LIN {X 0,Y 249.083,Z 81.458,A -85,B 0,C 180,E1 -19056.733,E2 -19056.733} C_VEL
LIN {X 0,Y 249.115,Z 81.452,A -85,B 0,C 180,E1 -19060.212,E2 -19060.212} C_VEL
LIN {X 0,Y 249.245,Z 81.417,A -85,B 0,C 180,E1 -19063.622,E2 -19063.622} C_VEL
LIN {X 0,Y 249.247,Z 81.438,A -85,B 0,C 180,E1 -19068.616,E2 -19068.616} C_VEL
LIN {X 0,Y 249.457,Z 81.409,A -85,B 0,C 180,E1 -19071.902,E2 -19071.902} C_VEL
LIN {X 0,Y 249.294,Z 81.412,A -85,B 0,C 180,E1 -19075.149,E2 -19075.149} C_VEL
LIN {X 0,Y 249.678,Z 81.38,A -85,B 0,C 180,E1 -19078.387,E2 -19078.387} C_VEL
LIN {X 0,Y 249.679,Z 81.385,A -85,B 0,C 180,E1 -19081.613,E2 -19081.613} C_VEL
LIN {X 0,Y 249.438,Z 81.412,A -85,B 0,C 180,E1 -19086.471,E2 -19086.471} C_VEL
LIN {X 0,Y 249.346,Z 81.422,A -85,B 0,C 180,E1 -19089.737,E2 -19089.737} C_VEL
LIN {X 0,Y 249.283,Z 81.427,A -85,B 0,C 180,E1 -19090.328,E2 -19090.328} C_VEL
LIN {X 0,Y 248.549,Z 81.525,A -85,B 0,C 180,E1 -19091.676,E2 -19091.676} C_VEL
LIN {X 0,Y 245.682,Z 81.88,A -85,B 0,C 180,E1 -19093.874,E2 -19093.874} C_VEL
LIN {X 0,Y 243.264,Z 82.181,A -85,B 0,C 180,E1 -19095.663,E2 -19095.663} C_VEL
LIN {X 0,Y 242.195,Z 82.315,A -85,B 0,C 180,E1 -19097.05,E2 -19097.05} C_VEL
LIN {X 0,Y 242.089,Z 82.325,A -85,B 0,C 180,E1 -19097.521,E2 -19097.521} C_VEL
LIN {X 0,Y 242.01,Z 82.339,A -85,B 0,C 180,E1 -19102.181,E2 -19102.181} C_VEL
LIN {X 0,Y 242.035,Z 82.335,A -85,B 0,C 180,E1 -19105.821,E2 -19105.821} C_VEL
LIN {X 0,Y 241.973,Z 82.344,A -85,B 0,C 180,E1 -19109.588,E2 -19109.588} C_VEL
LIN {X 0,Y 241.982,Z 82.343,A -85,B 0,C 180,E1 -19113.493,E2 -19113.493} C_VEL
LIN {X 0,Y 241.992,Z 82.341,A -85,B 0,C 180,E1 -19117.582,E2 -19117.582} C_VEL
LIN {X 0,Y 241.94,Z 82.348,A -85,B 0,C 180,E1 -19121.922,E2 -19121.922} C_VEL
LIN {X 0,Y 241.937,Z 82.351,A -85,B 0,C 180,E1 -19126.571,E2 -19126.571} C_VEL
LIN {X 0,Y 241.959,Z 82.347,A -85,B 0,C 180,E1 -19130.281,E2 -19130.281} C_VEL
LIN {X 0,Y 242.076,Z 82.527,A -85,B 0,C 180,E1 -19133.301,E2 -19133.301} C_VEL
LIN {X 0,Y 244.19,Z 91.874,A -85,B 0,C 180,E1 -19136.849,E2 -19136.849} C_VEL
LIN {X 0,Y 245.968,Z 100.654,A -85,B 0,C 180,E1 -19140.013,E2 -19140.013} C_VEL
LIN {X 0,Y 248.842,Z 109.122,A -85,B 0,C 180,E1 -19140.597,E2 -19140.597} C_VEL
LIN {X 0,Y 252.507,Z 138.269,A -85,B 0,C 180,E1 -19141.879,E2 -19141.879} C_VEL
LIN {X 0,Y 254.291,Z 157.169,A -85,B 0,C 180,E1 -19142.627,E2 -19142.627} C_VEL
LIN {X 0,Y 252.694,Z 210.32,A -85,B 0,C 180,E1 -19144.131,E2 -19144.131} C_VEL
LIN {X 0,Y 251.721,Z 223.453,A -85,B 0,C 180,E1 -19144.8,E2 -19144.8} C_VEL
LIN {X 0,Y 250.343,Z 236.124,A -85,B 0,C 180,E1 -19145.759,E2 -19145.759} C_VEL
LIN {X 0,Y 248.844,Z 247.387,A -85,B 0,C 180,E1 -19146.929,E2 -19146.929} C_VEL
LIN {X 0,Y 247.01,Z 259.074,A -85,B 0,C 180,E1 -19148.511,E2 -19148.511} C_VEL
LIN {X 0,Y 245.474,Z 268.522,A -85,B 0,C 180,E1 -19150.124,E2 -19150.124} C_VEL
LIN {X 0,Y 244.023,Z 276.962,A -85,B 0,C 180,E1 -19151.883,E2 -19151.883} C_VEL
LIN {X 0,Y 243.336,Z 280.982,A -85,B 0,C 180,E1 -19152.851,E2 -19152.851} C_VEL
LIN {X 0,Y 242.04,Z 289.578,A -85,B 0,C 180,E1 -19155.281,E2 -19155.281} C_VEL
LIN {X 0,Y 240.902,Z 296.619,A -85,B 0,C 180,E1 -19157.789,E2 -19157.789} C_VEL
LIN {X 0,Y 240.236,Z 303.085,A -85,B 0,C 180,E1 -19160.741,E2 -19160.741} C_VEL
LIN {X 0,Y 239.974,Z 307.313,A -85,B 0,C 180,E1 -19163.272,E2 -19163.272} C_VEL
LIN {X 0,Y 239.97,Z 309.546,A -85,B 0,C 180,E1 -19164.959,E2 -19164.959} C_VEL
LIN {X 0,Y 240.045,Z 311.282,A -85,B 0,C 180,E1 -19166.643,E2 -19166.643} C_VEL
LIN {X 0,Y 240.09,Z 312.593,A -85,B 0,C 180,E1 -19168.322,E2 -19168.322} C_VEL
LIN {X 0,Y 240.142,Z 313.499,A -85,B 0,C 180,E1 -19170,E2 -19170} C_VEL
LIN {X 0,Y 240.034,Z 313.985,A -85,B 0,C 180,E1 -19171.678,E2 -19171.678} C_VEL
LIN {X 0,Y 239.964,Z 314.036,A -85,B 0,C 180,E1 -19173.358,E2 -19173.358} C_VEL
LIN {X 0,Y 239.913,Z 313.67,A -85,B 0,C 180,E1 -19175.127,E2 -19175.127} C_VEL
LIN {X 0,Y 240.132,Z 311.863,A -85,B 0,C 180,E1 -19178.415,E2 -19178.415} C_VEL
LIN {X 0,Y 240.48,Z 310.31,A -85,B 0,C 180,E1 -19180.099,E2 -19180.099} C_VEL
LIN {X 0,Y 241.265,Z 307.21,A -85,B 0,C 180,E1 -19182.619,E2 -19182.619} C_VEL
LIN {X 0,Y 242.676,Z 303.085,A -85,B 0,C 180,E1 -19185.108,E2 -19185.108} C_VEL
LIN {X 0,Y 244.865,Z 296.801,A -85,B 0,C 180,E1 -19187.971,E2 -19187.971} C_VEL
LIN {X 0,Y 247.08,Z 289.994,A -85,B 0,C 180,E1 -19190.392,E2 -19190.392} C_VEL
LIN {X 0,Y 249.862,Z 281.575,A -85,B 0,C 180,E1 -19192.753,E2 -19192.753} C_VEL
LIN {X 0,Y 252.632,Z 272.932,A -85,B 0,C 180,E1 -19194.663,E2 -19194.663} C_VEL
LIN {X 0,Y 255.666,Z 262.319,A -85,B 0,C 180,E1 -19196.532,E2 -19196.532} C_VEL
LIN {X 0,Y 258.396,Z 251.803,A -85,B 0,C 180,E1 -19197.981,E2 -19197.981} C_VEL
LIN {X 0,Y 260.919,Z 240.172,A -85,B 0,C 180,E1 -19199.223,E2 -19199.223} C_VEL
LIN {X 0,Y 263.018,Z 228.115,A -85,B 0,C 180,E1 -19200.178,E2 -19200.178} C_VEL
LIN {X 0,Y 264.69,Z 214.429,A -85,B 0,C 180,E1 -19200.943,E2 -19200.943} C_VEL
LIN {X 0,Y 265.71,Z 200.941,A -85,B 0,C 180,E1 -19201.376,E2 -19201.376} C_VEL
LIN {X 0,Y 267.298,Z 160.216,A -85,B 0,C 180,E1 -19202.462,E2 -19202.462} C_VEL
LIN {X 0,Y 264.083,Z 138.448,A -85,B 0,C 180,E1 -19203.705,E2 -19203.705} C_VEL
LIN {X 0,Y 262.587,Z 131.019,A -85,B 0,C 180,E1 -19204.209,E2 -19204.209} C_VEL
LIN {X 0,Y 255.925,Z 116.639,A -85,B 0,C 180,E1 -19205.895,E2 -19205.895} C_VEL
LIN {X 0,Y 248.914,Z 103.116,A -85,B 0,C 180,E1 -19207.761,E2 -19207.761} C_VEL
LIN {X 0,Y 246.617,Z 98.7,A -85,B 0,C 180,E1 -19208.44,E2 -19208.44} C_VEL
LIN {X 0,Y 244.374,Z 90.616,A -85,B 0,C 180,E1 -19212.221,E2 -19212.221} C_VEL
LIN {X 0,Y 242.242,Z 83.517,A -85,B 0,C 180,E1 -19215.869,E2 -19215.869} C_VEL
LIN {X 0,Y 241.986,Z 82.334,A -85,B 0,C 180,E1 -19216.559,E2 -19216.559} C_VEL
LIN {X 0,Y 241.998,Z 82.337,A -85,B 0,C 180,E1 -19221.64,E2 -19221.64} C_VEL
LIN {X 0,Y 241.984,Z 82.339,A -85,B 0,C 180,E1 -19224.488,E2 -19224.488} C_VEL
LIN {X 0,Y 241.978,Z 82.344,A -85,B 0,C 180,E1 -19228.48,E2 -19228.48} C_VEL
LIN {X 0,Y 242.013,Z 82.34,A -85,B 0,C 180,E1 -19232.313,E2 -19232.313} C_VEL
LIN {X 0,Y 242.06,Z 82.333,A -85,B 0,C 180,E1 -19236.016,E2 -19236.016} C_VEL
LIN {X 0,Y 242.041,Z 82.33,A -85,B 0,C 180,E1 -19239.608,E2 -19239.608} C_VEL
LIN {X 0,Y 242.166,Z 82.307,A -85,B 0,C 180,E1 -19243.278,E2 -19243.278} C_VEL
LIN {X 0,Y 242.184,Z 82.304,A -85,B 0,C 180,E1 -19248.279,E2 -19248.279} C_VEL
LIN {X 0,Y 242.403,Z 82.284,A -85,B 0,C 180,E1 -19251.665,E2 -19251.665} C_VEL
LIN {X 0,Y 242.426,Z 82.271,A -85,B 0,C 180,E1 -19253.341,E2 -19253.341} C_VEL
LIN {X 0,Y 242.638,Z 82.246,A -85,B 0,C 180,E1 -19258.34,E2 -19258.34} C_VEL
LIN {X 0,Y 242.638,Z 82.26,A -85,B 0,C 180,E1 -19261.66,E2 -19261.66} C_VEL
LIN {X 0,Y 242.419,Z 82.288,A -85,B 0,C 180,E1 -19266.662,E2 -19266.662} C_VEL
LIN {X 0,Y 242.269,Z 82.298,A -85,B 0,C 180,E1 -19270.023,E2 -19270.023} C_VEL
LIN {X 0,Y 242.141,Z 82.315,A -85,B 0,C 180,E1 -19275.142,E2 -19275.142} C_VEL
LIN {X 0,Y 242.062,Z 82.321,A -85,B 0,C 180,E1 -19278.625,E2 -19278.625} C_VEL
LIN {X 0,Y 242.008,Z 82.333,A -85,B 0,C 180,E1 -19282.18,E2 -19282.18} C_VEL
LIN {X 0,Y 242.033,Z 82.335,A -85,B 0,C 180,E1 -19285.821,E2 -19285.821} C_VEL
LIN {X 0,Y 241.972,Z 82.343,A -85,B 0,C 180,E1 -19289.588,E2 -19289.588} C_VEL
LIN {X 0,Y 241.98,Z 82.338,A -85,B 0,C 180,E1 -19293.493,E2 -19293.493} C_VEL
LIN {X 0,Y 241.984,Z 82.339,A -85,B 0,C 180,E1 -19297.583,E2 -19297.583} C_VEL
LIN {X 0,Y 241.957,Z 82.325,A -85,B 0,C 180,E1 -19300.683,E2 -19300.683} C_VEL
LIN {X 0,Y 243.048,Z 85.314,A -85,B 0,C 180,E1 -19301.073,E2 -19301.073} C_VEL
LIN {X 0,Y 245.057,Z 87.692,A -85,B 0,C 180,E1 -19301.613,E2 -19301.613} C_VEL
LIN {X 0,Y 247.331,Z 91.154,A -85,B 0,C 180,E1 -19302.237,E2 -19302.237} C_VEL
LIN {X 0,Y 255.665,Z 104.188,A -85,B 0,C 180,E1 -19304.392,E2 -19304.392} C_VEL
LIN {X 0,Y 262.591,Z 116.027,A -85,B 0,C 180,E1 -19306.064,E2 -19306.064} C_VEL
LIN {X 0,Y 268.629,Z 128.906,A -85,B 0,C 180,E1 -19307.505,E2 -19307.505} C_VEL
LIN {X 0,Y 266.108,Z 185.116,A -85,B 0,C 180,E1 -19308.994,E2 -19308.994} C_VEL
LIN {X 0,Y 265.047,Z 197.91,A -85,B 0,C 180,E1 -19309.61,E2 -19309.61} C_VEL
LIN {X 0,Y 263.629,Z 209.846,A -85,B 0,C 180,E1 -19310.464,E2 -19310.464} C_VEL
LIN {X 0,Y 261.537,Z 222.38,A -85,B 0,C 180,E1 -19311.673,E2 -19311.673} C_VEL
LIN {X 0,Y 259.106,Z 233.731,A -85,B 0,C 180,E1 -19313.121,E2 -19313.121} C_VEL
LIN {X 0,Y 256.438,Z 244.411,A -85,B 0,C 180,E1 -19314.863,E2 -19314.863} C_VEL
LIN {X 0,Y 253.624,Z 253.941,A -85,B 0,C 180,E1 -19316.819,E2 -19316.819} C_VEL
LIN {X 0,Y 250.668,Z 263.079,A -85,B 0,C 180,E1 -19319.224,E2 -19319.224} C_VEL
LIN {X 0,Y 248.218,Z 269.982,A -85,B 0,C 180,E1 -19321.523,E2 -19321.523} C_VEL
LIN {X 0,Y 246.2,Z 275.278,A -85,B 0,C 180,E1 -19323.739,E2 -19323.739} C_VEL
LIN {X 0,Y 244.314,Z 279.989,A -85,B 0,C 180,E1 -19326.251,E2 -19326.251} C_VEL
LIN {X 0,Y 242.84,Z 283.543,A -85,B 0,C 180,E1 -19328.792,E2 -19328.792} C_VEL
LIN {X 0,Y 241.656,Z 286.048,A -85,B 0,C 180,E1 -19331.343,E2 -19331.343} C_VEL
LIN {X 0,Y 240.752,Z 287.793,A -85,B 0,C 180,E1 -19334.436,E2 -19334.436} C_VEL
LIN {X 0,Y 240.33,Z 288.182,A -85,B 0,C 180,E1 -19336.471,E2 -19336.471} C_VEL
LIN {X 0,Y 240.048,Z 288.099,A -85,B 0,C 180,E1 -19338.174,E2 -19338.174} C_VEL
LIN {X 0,Y 239.96,Z 287.599,A -85,B 0,C 180,E1 -19339.879,E2 -19339.879} C_VEL
LIN {X 0,Y 240.208,Z 285.348,A -85,B 0,C 180,E1 -19343.279,E2 -19343.279} C_VEL
LIN {X 0,Y 240.506,Z 282.58,A -85,B 0,C 180,E1 -19345.811,E2 -19345.811} C_VEL
LIN {X 0,Y 240.984,Z 278.805,A -85,B 0,C 180,E1 -19348.329,E2 -19348.329} C_VEL
LIN {X 0,Y 241.623,Z 273.927,A -85,B 0,C 180,E1 -19350.833,E2 -19350.833} C_VEL
LIN {X 0,Y 242.662,Z 267.78,A -85,B 0,C 180,E1 -19353.321,E2 -19353.321} C_VEL
LIN {X 0,Y 244.046,Z 260.126,A -85,B 0,C 180,E1 -19355.785,E2 -19355.785} C_VEL
LIN {X 0,Y 245.683,Z 250.533,A -85,B 0,C 180,E1 -19358.223,E2 -19358.223} C_VEL
LIN {X 0,Y 247.481,Z 240.605,A -85,B 0,C 180,E1 -19360.224,E2 -19360.224} C_VEL
LIN {X 0,Y 249.307,Z 229.377,A -85,B 0,C 180,E1 -19362,E2 -19362} C_VEL
LIN {X 0,Y 250.738,Z 218.415,A -85,B 0,C 180,E1 -19363.37,E2 -19363.37} C_VEL
LIN {X 0,Y 251.913,Z 206.317,A -85,B 0,C 180,E1 -19364.542,E2 -19364.542} C_VEL
LIN {X 0,Y 252.856,Z 193.622,A -85,B 0,C 180,E1 -19365.414,E2 -19365.414} C_VEL
LIN {X 0,Y 253.476,Z 180.26,A -85,B 0,C 180,E1 -19365.994,E2 -19365.994} C_VEL
LIN {X 0,Y 255.359,Z 113.557,A -85,B 0,C 180,E1 -19367.84,E2 -19367.84} C_VEL
LIN {X 0,Y 251.274,Z 102.48,A -85,B 0,C 180,E1 -19368.602,E2 -19368.602} C_VEL
LIN {X 0,Y 243.144,Z 85.322,A -85,B 0,C 180,E1 -19370.051,E2 -19370.051} C_VEL
LIN {X 0,Y 242.053,Z 82.327,A -85,B 0,C 180,E1 -19370.32,E2 -19370.32} C_VEL
LIN {X 0,Y 242.042,Z 82.334,A -85,B 0,C 180,E1 -19373.986,E2 -19373.986} C_VEL
LIN {X 0,Y 242.002,Z 82.341,A -85,B 0,C 180,E1 -19377.688,E2 -19377.688} C_VEL
LIN {X 0,Y 241.976,Z 82.341,A -85,B 0,C 180,E1 -19381.52,E2 -19381.52} C_VEL
LIN {X 0,Y 242.03,Z 82.338,A -85,B 0,C 180,E1 -19385.605,E2 -19385.605} C_VEL
LIN {X 0,Y 241.976,Z 82.344,A -85,B 0,C 180,E1 -19389.716,E2 -19389.716} C_VEL
LIN {X 0,Y 241.929,Z 82.346,A -85,B 0,C 180,E1 -19394.203,E2 -19394.203} C_VEL
LIN {X 0,Y 241.935,Z 82.345,A -85,B 0,C 180,E1 -19398.077,E2 -19398.077} C_VEL
LIN {X 0,Y 241.989,Z 82.339,A -85,B 0,C 180,E1 -19402.418,E2 -19402.418} C_VEL
LIN {X 0,Y 241.983,Z 82.34,A -85,B 0,C 180,E1 -19406.508,E2 -19406.508} C_VEL
LIN {X 0,Y 242.039,Z 82.332,A -85,B 0,C 180,E1 -19410.588,E2 -19410.588} C_VEL
LIN {X 0,Y 242.07,Z 82.329,A -85,B 0,C 180,E1 -19414.183,E2 -19414.183} C_VEL
LIN {X 0,Y 242.056,Z 82.334,A -85,B 0,C 180,E1 -19418.297,E2 -19418.297} C_VEL
LIN {X 0,Y 242.166,Z 82.298,A -85,B 0,C 180,E1 -19423.279,E2 -19423.279} C_VEL
LIN {X 0,Y 242.184,Z 82.317,A -85,B 0,C 180,E1 -19428.28,E2 -19428.28} C_VEL
LIN {X 0,Y 242.403,Z 82.288,A -85,B 0,C 180,E1 -19431.665,E2 -19431.665} C_VEL
LIN {X 0,Y 242.425,Z 82.278,A -85,B 0,C 180,E1 -19433.341,E2 -19433.341} C_VEL
LIN {X 0,Y 242.639,Z 82.255,A -85,B 0,C 180,E1 -19438.34,E2 -19438.34} C_VEL
LIN {X 0,Y 242.639,Z 82.262,A -85,B 0,C 180,E1 -19441.66,E2 -19441.66} C_VEL
LIN {X 0,Y 242.41,Z 82.288,A -85,B 0,C 180,E1 -19446.66,E2 -19446.66} C_VEL
LIN {X 0,Y 242.24,Z 82.305,A -85,B 0,C 180,E1 -19450.289,E2 -19450.289} C_VEL
LIN {X 0,Y 242.143,Z 82.321,A -85,B 0,C 180,E1 -19455.143,E2 -19455.143} C_VEL
LIN {X 0,Y 242.089,Z 82.325,A -85,B 0,C 180,E1 -19457.521,E2 -19457.521} C_VEL
LIN {X 0,Y 241.37,Z 82.42,A -85,B 0,C 180,E1 -19458.909,E2 -19458.909} C_VEL
LIN {X 0,Y 238.508,Z 82.777,A -85,B 0,C 180,E1 -19461.174,E2 -19461.174} C_VEL
LIN {X 0,Y 236.098,Z 83.079,A -85,B 0,C 180,E1 -19463.019,E2 -19463.019} C_VEL
LIN {X 0,Y 235.051,Z 83.206,A -85,B 0,C 180,E1 -19464.451,E2 -19464.451} C_VEL
LIN {X 0,Y 234.957,Z 83.216,A -85,B 0,C 180,E1 -19464.936,E2 -19464.936} C_VEL
LIN {X 0,Y 234.928,Z 83.222,A -85,B 0,C 180,E1 -19469.824,E2 -19469.824} C_VEL
LIN {X 0,Y 234.944,Z 83.221,A -85,B 0,C 180,E1 -19473.114,E2 -19473.114} C_VEL
LIN {X 0,Y 234.93,Z 83.223,A -85,B 0,C 180,E1 -19476.749,E2 -19476.749} C_VEL
LIN {X 0,Y 234.945,Z 83.219,A -85,B 0,C 180,E1 -19478.944,E2 -19478.944} C_VEL
LIN {X 0,Y 234.89,Z 83.224,A -85,B 0,C 180,E1 -19483.486,E2 -19483.486} C_VEL
LIN {X 0,Y 234.89,Z 83.229,A -85,B 0,C 180,E1 -19486.514,E2 -19486.514} C_VEL
LIN {X 0,Y 234.92,Z 83.224,A -85,B 0,C 180,E1 -19491.079,E2 -19491.079} C_VEL
LIN {X 0,Y 234.991,Z 83.34,A -85,B 0,C 180,E1 -19492.658,E2 -19492.658} C_VEL
LIN {X 0,Y 237.422,Z 93.969,A -85,B 0,C 180,E1 -19496.826,E2 -19496.826} C_VEL
LIN {X 0,Y 238.706,Z 100.362,A -85,B 0,C 180,E1 -19499.171,E2 -19499.171} C_VEL
LIN {X 0,Y 242.602,Z 111.238,A -85,B 0,C 180,E1 -19499.978,E2 -19499.978} C_VEL
LIN {X 0,Y 246.172,Z 140.741,A -85,B 0,C 180,E1 -19501.307,E2 -19501.307} C_VEL
LIN {X 0,Y 247.768,Z 157.118,A -85,B 0,C 180,E1 -19501.984,E2 -19501.984} C_VEL
LIN {X 0,Y 246.139,Z 209.645,A -85,B 0,C 180,E1 -19503.503,E2 -19503.503} C_VEL
LIN {X 0,Y 245.138,Z 222.877,A -85,B 0,C 180,E1 -19504.188,E2 -19504.188} C_VEL
LIN {X 0,Y 243.719,Z 235.602,A -85,B 0,C 180,E1 -19505.169,E2 -19505.169} C_VEL
LIN {X 0,Y 242.041,Z 247.703,A -85,B 0,C 180,E1 -19506.468,E2 -19506.468} C_VEL
LIN {X 0,Y 240.151,Z 259.261,A -85,B 0,C 180,E1 -19508.091,E2 -19508.091} C_VEL
LIN {X 0,Y 238.571,Z 268.612,A -85,B 0,C 180,E1 -19509.748,E2 -19509.748} C_VEL
LIN {X 0,Y 237,Z 277.213,A -85,B 0,C 180,E1 -19511.611,E2 -19511.611} C_VEL
LIN {X 0,Y 236.297,Z 281.517,A -85,B 0,C 180,E1 -19512.697,E2 -19512.697} C_VEL
LIN {X 0,Y 234.906,Z 290.102,A -85,B 0,C 180,E1 -19515.267,E2 -19515.267} C_VEL
LIN {X 0,Y 233.763,Z 296.97,A -85,B 0,C 180,E1 -19517.851,E2 -19517.851} C_VEL
LIN {X 0,Y 233.193,Z 302.47,A -85,B 0,C 180,E1 -19520.458,E2 -19520.458} C_VEL
LIN {X 0,Y 232.896,Z 306.752,A -85,B 0,C 180,E1 -19523.067,E2 -19523.067} C_VEL
LIN {X 0,Y 232.902,Z 309.02,A -85,B 0,C 180,E1 -19524.806,E2 -19524.806} C_VEL
LIN {X 0,Y 232.955,Z 310.795,A -85,B 0,C 180,E1 -19526.541,E2 -19526.541} C_VEL
LIN {X 0,Y 233.015,Z 312.131,A -85,B 0,C 180,E1 -19528.271,E2 -19528.271} C_VEL
LIN {X 0,Y 233.063,Z 313.059,A -85,B 0,C 180,E1 -19530,E2 -19530} C_VEL
LIN {X 0,Y 232.96,Z 313.578,A -85,B 0,C 180,E1 -19531.729,E2 -19531.729} C_VEL
LIN {X 0,Y 232.879,Z 313.662,A -85,B 0,C 180,E1 -19533.46,E2 -19533.46} C_VEL
LIN {X 0,Y 232.841,Z 313.344,A -85,B 0,C 180,E1 -19535.195,E2 -19535.195} C_VEL
LIN {X 0,Y 233.08,Z 311.558,A -85,B 0,C 180,E1 -19538.671,E2 -19538.671} C_VEL
LIN {X 0,Y 233.461,Z 310.048,A -85,B 0,C 180,E1 -19540.406,E2 -19540.406} C_VEL
LIN {X 0,Y 234.303,Z 306.995,A -85,B 0,C 180,E1 -19543.001,E2 -19543.001} C_VEL
LIN {X 0,Y 235.817,Z 302.92,A -85,B 0,C 180,E1 -19545.559,E2 -19545.559} C_VEL
LIN {X 0,Y 238.12,Z 296.696,A -85,B 0,C 180,E1 -19548.499,E2 -19548.499} C_VEL
LIN {X 0,Y 240.414,Z 289.955,A -85,B 0,C 180,E1 -19550.984,E2 -19550.984} C_VEL
LIN {X 0,Y 243.325,Z 281.632,A -85,B 0,C 180,E1 -19553.4,E2 -19553.4} C_VEL
LIN {X 0,Y 246.208,Z 273.103,A -85,B 0,C 180,E1 -19555.352,E2 -19555.352} C_VEL
LIN {X 0,Y 249.344,Z 262.609,A -85,B 0,C 180,E1 -19557.26,E2 -19557.26} C_VEL
LIN {X 0,Y 252.161,Z 252.24,A -85,B 0,C 180,E1 -19558.736,E2 -19558.736} C_VEL
LIN {X 0,Y 254.758,Z 240.886,A -85,B 0,C 180,E1 -19560.001,E2 -19560.001} C_VEL
LIN {X 0,Y 256.969,Z 229.22,A -85,B 0,C 180,E1 -19560.965,E2 -19560.965} C_VEL
LIN {X 0,Y 258.729,Z 215.521,A -85,B 0,C 180,E1 -19561.777,E2 -19561.777} C_VEL
LIN {X 0,Y 259.88,Z 202.343,A -85,B 0,C 180,E1 -19562.238,E2 -19562.238} C_VEL
LIN {X 0,Y 261.571,Z 161.244,A -85,B 0,C 180,E1 -19563.35,E2 -19563.35} C_VEL
LIN {X 0,Y 258.237,Z 138.412,A -85,B 0,C 180,E1 -19564.706,E2 -19564.706} C_VEL
LIN {X 0,Y 257.257,Z 134.015,A -85,B 0,C 180,E1 -19565.034,E2 -19565.034} C_VEL
LIN {X 0,Y 250.998,Z 120.403,A -85,B 0,C 180,E1 -19566.696,E2 -19566.696} C_VEL
LIN {X 0,Y 244.576,Z 107.852,A -85,B 0,C 180,E1 -19568.484,E2 -19568.484} C_VEL
LIN {X 0,Y 241.394,Z 102.28,A -85,B 0,C 180,E1 -19569.4,E2 -19569.4} C_VEL
LIN {X 0,Y 239.214,Z 98.113,A -85,B 0,C 180,E1 -19570.111,E2 -19570.111} C_VEL
LIN {X 0,Y 236.753,Z 89.25,A -85,B 0,C 180,E1 -19574.566,E2 -19574.566} C_VEL
LIN {X 0,Y 234.893,Z 83.215,A -85,B 0,C 180,E1 -19577.929,E2 -19577.929} C_VEL
LIN {X 0,Y 234.92,Z 83.213,A -85,B 0,C 180,E1 -19581.079,E2 -19581.079} C_VEL
LIN {X 0,Y 234.929,Z 83.216,A -85,B 0,C 180,E1 -19585.361,E2 -19585.361} C_VEL
LIN {X 0,Y 234.934,Z 83.213,A -85,B 0,C 180,E1 -19589.432,E2 -19589.432} C_VEL
LIN {X 0,Y 234.997,Z 83.202,A -85,B 0,C 180,E1 -19593.793,E2 -19593.793} C_VEL
LIN {X 0,Y 235.014,Z 83.2,A -85,B 0,C 180,E1 -19598.97,E2 -19598.97} C_VEL
LIN {X 0,Y 235.099,Z 83.186,A -85,B 0,C 180,E1 -19603.059,E2 -19603.059} C_VEL
LIN {X 0,Y 235.118,Z 83.183,A -85,B 0,C 180,E1 -19607.922,E2 -19607.922} C_VEL
LIN {X 0,Y 235.334,Z 83.167,A -85,B 0,C 180,E1 -19611.412,E2 -19611.412} C_VEL
LIN {X 0,Y 235.376,Z 83.149,A -85,B 0,C 180,E1 -19613.14,E2 -19613.14} C_VEL
LIN {X 0,Y 235.597,Z 83.122,A -85,B 0,C 180,E1 -19618.29,E2 -19618.29} C_VEL
LIN {X 0,Y 235.598,Z 83.136,A -85,B 0,C 180,E1 -19621.709,E2 -19621.709} C_VEL
LIN {X 0,Y 235.37,Z 83.167,A -85,B 0,C 180,E1 -19626.859,E2 -19626.859} C_VEL
LIN {X 0,Y 235.216,Z 83.179,A -85,B 0,C 180,E1 -19630.327,E2 -19630.327} C_VEL
LIN {X 0,Y 235.095,Z 83.197,A -85,B 0,C 180,E1 -19635.607,E2 -19635.607} C_VEL
LIN {X 0,Y 235.002,Z 83.201,A -85,B 0,C 180,E1 -19639.206,E2 -19639.206} C_VEL
LIN {X 0,Y 234.953,Z 83.208,A -85,B 0,C 180,E1 -19642.883,E2 -19642.883} C_VEL
LIN {X 0,Y 234.948,Z 83.21,A -85,B 0,C 180,E1 -19646.66,E2 -19646.66} C_VEL
LIN {X 0,Y 234.901,Z 83.217,A -85,B 0,C 180,E1 -19650.572,E2 -19650.572} C_VEL
LIN {X 0,Y 234.926,Z 83.217,A -85,B 0,C 180,E1 -19654.638,E2 -19654.638} C_VEL
LIN {X 0,Y 234.925,Z 83.216,A -85,B 0,C 180,E1 -19659.031,E2 -19659.031} C_VEL
LIN {X 0,Y 235.989,Z 86.175,A -85,B 0,C 180,E1 -19659.453,E2 -19659.453} C_VEL
LIN {X 0,Y 238.055,Z 88.413,A -85,B 0,C 180,E1 -19660.046,E2 -19660.046} C_VEL
LIN {X 0,Y 239.918,Z 91.502,A -85,B 0,C 180,E1 -19660.612,E2 -19660.612} C_VEL
LIN {X 0,Y 241.752,Z 94.11,A -85,B 0,C 180,E1 -19661.136,E2 -19661.136} C_VEL
LIN {X 0,Y 248.766,Z 104.769,A -85,B 0,C 180,E1 -19663.056,E2 -19663.056} C_VEL
LIN {X 0,Y 256.888,Z 118.447,A -85,B 0,C 180,E1 -19665.133,E2 -19665.133} C_VEL
LIN {X 0,Y 262.926,Z 131.138,A -85,B 0,C 180,E1 -19666.639,E2 -19666.639} C_VEL
LIN {X 0,Y 260.28,Z 186.314,A -85,B 0,C 180,E1 -19668.129,E2 -19668.129} C_VEL
LIN {X 0,Y 259.08,Z 199.617,A -85,B 0,C 180,E1 -19668.801,E2 -19668.801} C_VEL
LIN {X 0,Y 257.583,Z 211.623,A -85,B 0,C 180,E1 -19669.711,E2 -19669.711} C_VEL
LIN {X 0,Y 255.648,Z 222.43,A -85,B 0,C 180,E1 -19670.78,E2 -19670.78} C_VEL
LIN {X 0,Y 252.995,Z 234.347,A -85,B 0,C 180,E1 -19672.328,E2 -19672.328} C_VEL
LIN {X 0,Y 250.513,Z 243.897,A -85,B 0,C 180,E1 -19673.904,E2 -19673.904} C_VEL
LIN {X 0,Y 247.573,Z 253.623,A -85,B 0,C 180,E1 -19675.899,E2 -19675.899} C_VEL
LIN {X 0,Y 244.894,Z 261.521,A -85,B 0,C 180,E1 -19677.933,E2 -19677.933} C_VEL
LIN {X 0,Y 242.122,Z 269.178,A -85,B 0,C 180,E1 -19680.432,E2 -19680.432} C_VEL
LIN {X 0,Y 239.67,Z 275.284,A -85,B 0,C 180,E1 -19682.966,E2 -19682.966} C_VEL
LIN {X 0,Y 237.658,Z 280.076,A -85,B 0,C 180,E1 -19685.543,E2 -19685.543} C_VEL
LIN {X 0,Y 236.077,Z 283.706,A -85,B 0,C 180,E1 -19688.153,E2 -19688.153} C_VEL
LIN {X 0,Y 234.795,Z 286.284,A -85,B 0,C 180,E1 -19690.776,E2 -19690.776} C_VEL
LIN {X 0,Y 234.159,Z 287.477,A -85,B 0,C 180,E1 -19692.534,E2 -19692.534} C_VEL
LIN {X 0,Y 233.706,Z 288.219,A -85,B 0,C 180,E1 -19694.297,E2 -19694.297} C_VEL
LIN {X 0,Y 233.303,Z 288.555,A -85,B 0,C 180,E1 -19696.055,E2 -19696.055} C_VEL
LIN {X 0,Y 232.886,Z 288.062,A -85,B 0,C 180,E1 -19699.568,E2 -19699.568} C_VEL
LIN {X 0,Y 232.898,Z 287.179,A -85,B 0,C 180,E1 -19701.322,E2 -19701.322} C_VEL
LIN {X 0,Y 233.261,Z 285.191,A -85,B 0,C 180,E1 -19703.863,E2 -19703.863} C_VEL
LIN {X 0,Y 233.481,Z 282.097,A -85,B 0,C 180,E1 -19706.549,E2 -19706.549} C_VEL
LIN {X 0,Y 234.078,Z 278.038,A -85,B 0,C 180,E1 -19709.14,E2 -19709.14} C_VEL
LIN {X 0,Y 234.999,Z 271.83,A -85,B 0,C 180,E1 -19712.143,E2 -19712.143} C_VEL
LIN {X 0,Y 236.318,Z 265.058,A -85,B 0,C 180,E1 -19714.691,E2 -19714.691} C_VEL
LIN {X 0,Y 237.821,Z 256.654,A -85,B 0,C 180,E1 -19717.215,E2 -19717.215} C_VEL
LIN {X 0,Y 239.351,Z 248.004,A -85,B 0,C 180,E1 -19719.294,E2 -19719.294} C_VEL
LIN {X 0,Y 241.391,Z 237.309,A -85,B 0,C 180,E1 -19721.334,E2 -19721.334} C_VEL
LIN {X 0,Y 243.057,Z 226.683,A -85,B 0,C 180,E1 -19722.95,E2 -19722.95} C_VEL
LIN {X 0,Y 244.524,Z 214.816,A -85,B 0,C 180,E1 -19724.353,E2 -19724.353} C_VEL
LIN {X 0,Y 245.663,Z 202.504,A -85,B 0,C 180,E1 -19725.451,E2 -19725.451} C_VEL
LIN {X 0,Y 246.537,Z 189.774,A -85,B 0,C 180,E1 -19726.244,E2 -19726.244} C_VEL
LIN {X 0,Y 247.087,Z 175.916,A -85,B 0,C 180,E1 -19726.75,E2 -19726.75} C_VEL
LIN {X 0,Y 248.886,Z 115.206,A -85,B 0,C 180,E1 -19728.459,E2 -19728.459} C_VEL
LIN {X 0,Y 245.313,Z 105.535,A -85,B 0,C 180,E1 -19729.153,E2 -19729.153} C_VEL
LIN {X 0,Y 237.664,Z 89.241,A -85,B 0,C 180,E1 -19730.575,E2 -19730.575} C_VEL
LIN {X 0,Y 235.1,Z 83.875,A -85,B 0,C 180,E1 -19731.072,E2 -19731.072} C_VEL
LIN {X 0,Y 234.999,Z 83.205,A -85,B 0,C 180,E1 -19731.152,E2 -19731.152} C_VEL
LIN {X 0,Y 234.995,Z 83.214,A -85,B 0,C 180,E1 -19736.206,E2 -19736.206} C_VEL
LIN {X 0,Y 234.924,Z 83.22,A -85,B 0,C 180,E1 -19740.569,E2 -19740.569} C_VEL
LIN {X 0,Y 234.962,Z 83.216,A -85,B 0,C 180,E1 -19744.633,E2 -19744.633} C_VEL
LIN {X 0,Y 234.943,Z 83.218,A -85,B 0,C 180,E1 -19748.945,E2 -19748.945} C_VEL
LIN {X 0,Y 234.888,Z 83.227,A -85,B 0,C 180,E1 -19753.486,E2 -19753.486} C_VEL
LIN {X 0,Y 234.882,Z 83.223,A -85,B 0,C 180,E1 -19756.513,E2 -19756.513} C_VEL
LIN {X 0,Y 234.92,Z 83.219,A -85,B 0,C 180,E1 -19761.079,E2 -19761.079} C_VEL
LIN {X 0,Y 234.929,Z 83.219,A -85,B 0,C 180,E1 -19765.362,E2 -19765.362} C_VEL
LIN {X 0,Y 234.934,Z 83.215,A -85,B 0,C 180,E1 -19769.433,E2 -19769.433} C_VEL
LIN {X 0,Y 234.997,Z 83.21,A -85,B 0,C 180,E1 -19773.794,E2 -19773.794} C_VEL
LIN {X 0,Y 235.015,Z 83.209,A -85,B 0,C 180,E1 -19778.97,E2 -19778.97} C_VEL
LIN {X 0,Y 235.1,Z 83.177,A -85,B 0,C 180,E1 -19783.06,E2 -19783.06} C_VEL
LIN {X 0,Y 235.118,Z 83.195,A -85,B 0,C 180,E1 -19787.922,E2 -19787.922} C_VEL
LIN {X 0,Y 235.334,Z 83.168,A -85,B 0,C 180,E1 -19791.413,E2 -19791.413} C_VEL
LIN {X 0,Y 235.376,Z 83.156,A -85,B 0,C 180,E1 -19793.141,E2 -19793.141} C_VEL
LIN {X 0,Y 235.598,Z 83.131,A -85,B 0,C 180,E1 -19798.291,E2 -19798.291} C_VEL
LIN {X 0,Y 235.598,Z 83.14,A -85,B 0,C 180,E1 -19801.71,E2 -19801.71} C_VEL
LIN {X 0,Y 235.361,Z 83.166,A -85,B 0,C 180,E1 -19806.86,E2 -19806.86} C_VEL
LIN {X 0,Y 235.215,Z 83.18,A -85,B 0,C 180,E1 -19810.328,E2 -19810.328} C_VEL
LIN {X 0,Y 235.097,Z 83.198,A -85,B 0,C 180,E1 -19815.608,E2 -19815.608} C_VEL
LIN {X 0,Y 235.003,Z 83.211,A -85,B 0,C 180,E1 -19819.206,E2 -19819.206} C_VEL
LIN {X 0,Y 234.955,Z 83.22,A -85,B 0,C 180,E1 -19822.884,E2 -19822.884} C_VEL
LIN {X 0,Y 234.957,Z 83.216,A -85,B 0,C 180,E1 -19824.936,E2 -19824.936} C_VEL
LIN {X 0,Y 234.256,Z 83.306,A -85,B 0,C 180,E1 -19826.367,E2 -19826.367} C_VEL
LIN {X 0,Y 231.369,Z 83.667,A -85,B 0,C 180,E1 -19828.701,E2 -19828.701} C_VEL
LIN {X 0,Y 228.941,Z 83.97,A -85,B 0,C 180,E1 -19830.605,E2 -19830.605} C_VEL
LIN {X 0,Y 227.913,Z 84.097,A -85,B 0,C 180,E1 -19832.083,E2 -19832.083} C_VEL
LIN {X 0,Y 227.835,Z 84.101,A -85,B 0,C 180,E1 -19832.584,E2 -19832.584} C_VEL
LIN {X 0,Y 227.895,Z 84.1,A -85,B 0,C 180,E1 -19836.696,E2 -19836.696} C_VEL
LIN {X 0,Y 227.829,Z 84.108,A -85,B 0,C 180,E1 -19840.377,E2 -19840.377} C_VEL
LIN {X 0,Y 227.836,Z 84.104,A -85,B 0,C 180,E1 -19845.193,E2 -19845.193} C_VEL
LIN {X 0,Y 227.829,Z 84.108,A -85,B 0,C 180,E1 -19849.623,E2 -19849.623} C_VEL
LIN {X 0,Y 227.944,Z 84.265,A -85,B 0,C 180,E1 -19852.02,E2 -19852.02} C_VEL
LIN {X 0,Y 230.383,Z 94.817,A -85,B 0,C 180,E1 -19856.32,E2 -19856.32} C_VEL
LIN {X 0,Y 231.402,Z 99.861,A -85,B 0,C 180,E1 -19858.256,E2 -19858.256} C_VEL
LIN {X 0,Y 236.351,Z 113.094,A -85,B 0,C 180,E1 -19859.314,E2 -19859.314} C_VEL
LIN {X 0,Y 239.765,Z 142.084,A -85,B 0,C 180,E1 -19860.66,E2 -19860.66} C_VEL
LIN {X 0,Y 241.258,Z 158.328,A -85,B 0,C 180,E1 -19861.347,E2 -19861.347} C_VEL
LIN {X 0,Y 239.614,Z 208.938,A -85,B 0,C 180,E1 -19862.841,E2 -19862.841} C_VEL
LIN {X 0,Y 238.595,Z 222.285,A -85,B 0,C 180,E1 -19863.543,E2 -19863.543} C_VEL
LIN {X 0,Y 237.131,Z 235.067,A -85,B 0,C 180,E1 -19864.548,E2 -19864.548} C_VEL
LIN {X 0,Y 235.554,Z 246.424,A -85,B 0,C 180,E1 -19865.779,E2 -19865.779} C_VEL
LIN {X 0,Y 233.464,Z 258.128,A -85,B 0,C 180,E1 -19867.429,E2 -19867.429} C_VEL
LIN {X 0,Y 231.679,Z 268.702,A -85,B 0,C 180,E1 -19869.351,E2 -19869.351} C_VEL
LIN {X 0,Y 230.081,Z 277.151,A -85,B 0,C 180,E1 -19871.249,E2 -19871.249} C_VEL
LIN {X 0,Y 229.37,Z 280.655,A -85,B 0,C 180,E1 -19872.157,E2 -19872.157} C_VEL
LIN {X 0,Y 228.166,Z 288.037,A -85,B 0,C 180,E1 -19874.364,E2 -19874.364} C_VEL
LIN {X 0,Y 226.972,Z 295.274,A -85,B 0,C 180,E1 -19877.027,E2 -19877.027} C_VEL
LIN {X 0,Y 226.169,Z 301.857,A -85,B 0,C 180,E1 -19880.159,E2 -19880.159} C_VEL
LIN {X 0,Y 225.82,Z 306.19,A -85,B 0,C 180,E1 -19882.849,E2 -19882.849} C_VEL
LIN {X 0,Y 225.809,Z 308.73,A -85,B 0,C 180,E1 -19884.85,E2 -19884.85} C_VEL
LIN {X 0,Y 225.869,Z 310.309,A -85,B 0,C 180,E1 -19886.432,E2 -19886.432} C_VEL
LIN {X 0,Y 225.941,Z 311.668,A -85,B 0,C 180,E1 -19888.217,E2 -19888.217} C_VEL
LIN {X 0,Y 225.987,Z 312.619,A -85,B 0,C 180,E1 -19890,E2 -19890} C_VEL
LIN {X 0,Y 225.887,Z 313.162,A -85,B 0,C 180,E1 -19891.783,E2 -19891.783} C_VEL
LIN {X 0,Y 225.774,Z 313.084,A -85,B 0,C 180,E1 -19895.05,E2 -19895.05} C_VEL
LIN {X 0,Y 225.763,Z 312.31,A -85,B 0,C 180,E1 -19897.153,E2 -19897.153} C_VEL
LIN {X 0,Y 226.024,Z 311.249,A -85,B 0,C 180,E1 -19898.944,E2 -19898.944} C_VEL
LIN {X 0,Y 226.439,Z 309.784,A -85,B 0,C 180,E1 -19900.732,E2 -19900.732} C_VEL
LIN {X 0,Y 227.363,Z 306.772,A -85,B 0,C 180,E1 -19903.405,E2 -19903.405} C_VEL
LIN {X 0,Y 228.974,Z 302.746,A -85,B 0,C 180,E1 -19906.036,E2 -19906.036} C_VEL
LIN {X 0,Y 231.392,Z 296.601,A -85,B 0,C 180,E1 -19909.057,E2 -19909.057} C_VEL
LIN {X 0,Y 233.763,Z 289.925,A -85,B 0,C 180,E1 -19911.61,E2 -19911.61} C_VEL
LIN {X 0,Y 236.831,Z 281.675,A -85,B 0,C 180,E1 -19914.081,E2 -19914.081} C_VEL
LIN {X 0,Y 239.812,Z 273.259,A -85,B 0,C 180,E1 -19916.078,E2 -19916.078} C_VEL
LIN {X 0,Y 243.08,Z 262.899,A -85,B 0,C 180,E1 -19918.023,E2 -19918.023} C_VEL
LIN {X 0,Y 245.975,Z 252.676,A -85,B 0,C 180,E1 -19919.529,E2 -19919.529} C_VEL
LIN {X 0,Y 248.654,Z 241.52,A -85,B 0,C 180,E1 -19920.816,E2 -19920.816} C_VEL
LIN {X 0,Y 251.147,Z 229.038,A -85,B 0,C 180,E1 -19921.883,E2 -19921.883} C_VEL
LIN {X 0,Y 252.918,Z 215.886,A -85,B 0,C 180,E1 -19922.684,E2 -19922.684} C_VEL
LIN {X 0,Y 254.159,Z 202.363,A -85,B 0,C 180,E1 -19923.178,E2 -19923.178} C_VEL
LIN {X 0,Y 255.834,Z 161.301,A -85,B 0,C 180,E1 -19924.326,E2 -19924.326} C_VEL
LIN {X 0,Y 252.374,Z 137.934,A -85,B 0,C 180,E1 -19925.789,E2 -19925.789} C_VEL
LIN {X 0,Y 246.311,Z 124.511,A -85,B 0,C 180,E1 -19927.479,E2 -19927.479} C_VEL
LIN {X 0,Y 240.097,Z 112.246,A -85,B 0,C 180,E1 -19929.289,E2 -19929.289} C_VEL
LIN {X 0,Y 234.614,Z 102.494,A -85,B 0,C 180,E1 -19930.973,E2 -19930.973} C_VEL
LIN {X 0,Y 231.999,Z 98.038,A -85,B 0,C 180,E1 -19931.815,E2 -19931.815} C_VEL
LIN {X 0,Y 231.797,Z 97.488,A -85,B 0,C 180,E1 -19931.966,E2 -19931.966} C_VEL
LIN {X 0,Y 230.001,Z 91.127,A -85,B 0,C 180,E1 -19935.348,E2 -19935.348} C_VEL
LIN {X 0,Y 227.837,Z 84.093,A -85,B 0,C 180,E1 -19939.518,E2 -19939.518} C_VEL
LIN {X 0,Y 227.882,Z 84.091,A -85,B 0,C 180,E1 -19944.128,E2 -19944.128} C_VEL
LIN {X 0,Y 227.873,Z 84.1,A -85,B 0,C 180,E1 -19948.378,E2 -19948.378} C_VEL
LIN {X 0,Y 227.889,Z 84.098,A -85,B 0,C 180,E1 -19952.445,E2 -19952.445} C_VEL
LIN {X 0,Y 227.917,Z 84.096,A -85,B 0,C 180,E1 -19956.367,E2 -19956.367} C_VEL
LIN {X 0,Y 227.946,Z 84.09,A -85,B 0,C 180,E1 -19960.175,E2 -19960.175} C_VEL
LIN {X 0,Y 228.061,Z 84.066,A -85,B 0,C 180,E1 -19963.898,E2 -19963.898} C_VEL
LIN {X 0,Y 228.076,Z 84.061,A -85,B 0,C 180,E1 -19967.543,E2 -19967.543} C_VEL
LIN {X 0,Y 228.271,Z 84.05,A -85,B 0,C 180,E1 -19971.144,E2 -19971.144} C_VEL
LIN {X 0,Y 228.327,Z 84.027,A -85,B 0,C 180,E1 -19972.927,E2 -19972.927} C_VEL
LIN {X 0,Y 228.556,Z 83.999,A -85,B 0,C 180,E1 -19978.238,E2 -19978.238} C_VEL
LIN {X 0,Y 228.556,Z 84.012,A -85,B 0,C 180,E1 -19981.762,E2 -19981.762} C_VEL
LIN {X 0,Y 228.321,Z 84.042,A -85,B 0,C 180,E1 -19987.072,E2 -19987.072} C_VEL
LIN {X 0,Y 228.147,Z 84.064,A -85,B 0,C 180,E1 -19990.651,E2 -19990.651} C_VEL
LIN {X 0,Y 228.052,Z 84.064,A -85,B 0,C 180,E1 -19994.273,E2 -19994.273} C_VEL
LIN {X 0,Y 228,Z 84.074,A -85,B 0,C 180,E1 -19997.953,E2 -19997.953} C_VEL
LIN {X 0,Y 227.925,Z 84.085,A -85,B 0,C 180,E1 -20002.325,E2 -20002.325} C_VEL
LIN {X 0,Y 227.925,Z 84.085,A -85,B 0,C 180,E1 -20006.593,E2 -20006.593} C_VEL
LIN {X 0,Y 227.875,Z 84.093,A -85,B 0,C 180,E1 -20010.281,E2 -20010.281} C_VEL
LIN {X 0,Y 227.877,Z 84.093,A -85,B 0,C 180,E1 -20013.72,E2 -20013.72} C_VEL
LIN {X 0,Y 227.876,Z 84.198,A -85,B 0,C 180,E1 -20017.262,E2 -20017.262} C_VEL
LIN {X 0,Y 228.761,Z 86.793,A -85,B 0,C 180,E1 -20017.622,E2 -20017.622} C_VEL
LIN {X 0,Y 230.744,Z 88.982,A -85,B 0,C 180,E1 -20018.247,E2 -20018.247} C_VEL
LIN {X 0,Y 233.547,Z 93.094,A -85,B 0,C 180,E1 -20019.145,E2 -20019.145} C_VEL
LIN {X 0,Y 239.991,Z 102.481,A -85,B 0,C 180,E1 -20021.077,E2 -20021.077} C_VEL
LIN {X 0,Y 248.414,Z 115.987,A -85,B 0,C 180,E1 -20023.41,E2 -20023.41} C_VEL
LIN {X 0,Y 253.828,Z 125.97,A -85,B 0,C 180,E1 -20024.835,E2 -20024.835} C_VEL
LIN {X 0,Y 257.179,Z 133.207,A -85,B 0,C 180,E1 -20025.71,E2 -20025.71} C_VEL
LIN {X 0,Y 254.619,Z 186.261,A -85,B 0,C 180,E1 -20027.175,E2 -20027.175} C_VEL
LIN {X 0,Y 253.469,Z 199.007,A -85,B 0,C 180,E1 -20027.817,E2 -20027.817} C_VEL
LIN {X 0,Y 251.882,Z 211.186,A -85,B 0,C 180,E1 -20028.728,E2 -20028.728} C_VEL
LIN {X 0,Y 249.698,Z 223.11,A -85,B 0,C 180,E1 -20029.921,E2 -20029.921} C_VEL
LIN {X 0,Y 246.933,Z 234.964,A -85,B 0,C 180,E1 -20031.494,E2 -20031.494} C_VEL
LIN {X 0,Y 244.068,Z 245.45,A -85,B 0,C 180,E1 -20033.282,E2 -20033.282} C_VEL
LIN {X 0,Y 240.981,Z 255.004,A -85,B 0,C 180,E1 -20035.34,E2 -20035.34} C_VEL
LIN {X 0,Y 237.736,Z 264.09,A -85,B 0,C 180,E1 -20037.851,E2 -20037.851} C_VEL
LIN {X 0,Y 235.332,Z 270.27,A -85,B 0,C 180,E1 -20040.004,E2 -20040.004} C_VEL
LIN {X 0,Y 232.432,Z 277.074,A -85,B 0,C 180,E1 -20043.028,E2 -20043.028} C_VEL
LIN {X 0,Y 230.364,Z 281.662,A -85,B 0,C 180,E1 -20045.774,E2 -20045.774} C_VEL
LIN {X 0,Y 228.83,Z 284.88,A -85,B 0,C 180,E1 -20048.374,E2 -20048.374} C_VEL
LIN {X 0,Y 227.953,Z 286.522,A -85,B 0,C 180,E1 -20050.176,E2 -20050.176} C_VEL
LIN {X 0,Y 227.231,Z 287.751,A -85,B 0,C 180,E1 -20051.984,E2 -20051.984} C_VEL
LIN {X 0,Y 226.675,Z 288.604,A -85,B 0,C 180,E1 -20053.976,E2 -20053.976} C_VEL
LIN {X 0,Y 225.976,Z 288.911,A -85,B 0,C 180,E1 -20057.426,E2 -20057.426} C_VEL
LIN {X 0,Y 225.809,Z 288.505,A -85,B 0,C 180,E1 -20059.237,E2 -20059.237} C_VEL
LIN {X 0,Y 225.813,Z 287.684,A -85,B 0,C 180,E1 -20061.048,E2 -20061.048} C_VEL
LIN {X 0,Y 226.172,Z 285.522,A -85,B 0,C 180,E1 -20063.91,E2 -20063.91} C_VEL
LIN {X 0,Y 226.396,Z 282.727,A -85,B 0,C 180,E1 -20066.441,E2 -20066.441} C_VEL
LIN {X 0,Y 226.979,Z 278.744,A -85,B 0,C 180,E1 -20069.113,E2 -20069.113} C_VEL
LIN {X 0,Y 227.904,Z 272.634,A -85,B 0,C 180,E1 -20072.209,E2 -20072.209} C_VEL
LIN {X 0,Y 229.262,Z 265.952,A -85,B 0,C 180,E1 -20074.836,E2 -20074.836} C_VEL
LIN {X 0,Y 230.802,Z 257.692,A -85,B 0,C 180,E1 -20077.436,E2 -20077.436} C_VEL
LIN {X 0,Y 232.394,Z 249.19,A -85,B 0,C 180,E1 -20079.575,E2 -20079.575} C_VEL
LIN {X 0,Y 234.301,Z 239.822,A -85,B 0,C 180,E1 -20081.462,E2 -20081.462} C_VEL
LIN {X 0,Y 236.212,Z 228.243,A -85,B 0,C 180,E1 -20083.332,E2 -20083.332} C_VEL
LIN {X 0,Y 237.744,Z 216.811,A -85,B 0,C 180,E1 -20084.772,E2 -20084.772} C_VEL
LIN {X 0,Y 238.905,Z 205.009,A -85,B 0,C 180,E1 -20085.9,E2 -20085.9} C_VEL
LIN {X 0,Y 239.924,Z 191.365,A -85,B 0,C 180,E1 -20086.814,E2 -20086.814} C_VEL
LIN {X 0,Y 240.508,Z 177.857,A -85,B 0,C 180,E1 -20087.355,E2 -20087.355} C_VEL
LIN {X 0,Y 242.418,Z 116.804,A -85,B 0,C 180,E1 -20089.115,E2 -20089.115} C_VEL
LIN {X 0,Y 239.268,Z 108.327,A -85,B 0,C 180,E1 -20089.752,E2 -20089.752} C_VEL
LIN {X 0,Y 232,Z 92.831,A -85,B 0,C 180,E1 -20091.16,E2 -20091.16} C_VEL
LIN {X 0,Y 228.168,Z 85.142,A -85,B 0,C 180,E1 -20091.928,E2 -20091.928} C_VEL
LIN {X 0,Y 227.958,Z 84.087,A -85,B 0,C 180,E1 -20092.006,E2 -20092.006} C_VEL
LIN {X 0,Y 227.943,Z 84.092,A -85,B 0,C 180,E1 -20096.602,E2 -20096.602} C_VEL
LIN {X 0,Y 227.898,Z 84.096,A -85,B 0,C 180,E1 -20100.291,E2 -20100.291} C_VEL
LIN {X 0,Y 227.891,Z 84.097,A -85,B 0,C 180,E1 -20103.719,E2 -20103.719} C_VEL
LIN {X 0,Y 227.871,Z 84.1,A -85,B 0,C 180,E1 -20108.086,E2 -20108.086} C_VEL
LIN {X 0,Y 227.816,Z 84.105,A -85,B 0,C 180,E1 -20112.742,E2 -20112.742} C_VEL
LIN {X 0,Y 227.808,Z 84.107,A -85,B 0,C 180,E1 -20117.257,E2 -20117.257} C_VEL
LIN {X 0,Y 227.846,Z 84.101,A -85,B 0,C 180,E1 -20121.909,E2 -20121.909} C_VEL
LIN {X 0,Y 227.881,Z 84.096,A -85,B 0,C 180,E1 -20126.378,E2 -20126.378} C_VEL
LIN {X 0,Y 227.922,Z 84.089,A -85,B 0,C 180,E1 -20130.438,E2 -20130.438} C_VEL
LIN {X 0,Y 227.932,Z 84.09,A -85,B 0,C 180,E1 -20134.426,E2 -20134.426} C_VEL
LIN {X 0,Y 227.965,Z 84.089,A -85,B 0,C 180,E1 -20138.288,E2 -20138.288} C_VEL
LIN {X 0,Y 228.038,Z 84.057,A -85,B 0,C 180,E1 -20142.826,E2 -20142.826} C_VEL
LIN {X 0,Y 228.076,Z 84.07,A -85,B 0,C 180,E1 -20147.544,E2 -20147.544} C_VEL
LIN {X 0,Y 228.27,Z 84.047,A -85,B 0,C 180,E1 -20151.145,E2 -20151.145} C_VEL
LIN {X 0,Y 228.326,Z 84.033,A -85,B 0,C 180,E1 -20152.928,E2 -20152.928} C_VEL
LIN {X 0,Y 228.557,Z 84.006,A -85,B 0,C 180,E1 -20158.238,E2 -20158.238} C_VEL
LIN {X 0,Y 228.557,Z 84.017,A -85,B 0,C 180,E1 -20161.762,E2 -20161.762} C_VEL
LIN {X 0,Y 228.313,Z 84.045,A -85,B 0,C 180,E1 -20167.073,E2 -20167.073} C_VEL
LIN {X 0,Y 228.146,Z 84.06,A -85,B 0,C 180,E1 -20170.651,E2 -20170.651} C_VEL
LIN {X 0,Y 228.047,Z 84.075,A -85,B 0,C 180,E1 -20176.103,E2 -20176.103} C_VEL
LIN {X 0,Y 227.936,Z 84.088,A -85,B 0,C 180,E1 -20179.826,E2 -20179.826} C_VEL
LIN {X 0,Y 227.903,Z 84.096,A -85,B 0,C 180,E1 -20183.634,E2 -20183.634} C_VEL
LIN {X 0,Y 227.861,Z 84.102,A -85,B 0,C 180,E1 -20187.559,E2 -20187.559} C_VEL
LIN {X 0,Y 227.859,Z 84.103,A -85,B 0,C 180,E1 -20191.624,E2 -20191.624} C_VEL
LIN {X 0,Y 227.835,Z 84.101,A -85,B 0,C 180,E1 -20192.584,E2 -20192.584} C_VEL
LIN {X 0,Y 227.194,Z 84.186,A -85,B 0,C 180,E1 -20194.059,E2 -20194.059} C_VEL
LIN {X 0,Y 224.385,Z 84.539,A -85,B 0,C 180,E1 -20196.468,E2 -20196.468} C_VEL
LIN {X 0,Y 221.133,Z 84.943,A -85,B 0,C 180,E1 -20199.443,E2 -20199.443} C_VEL
LIN {X 0,Y 220.78,Z 84.983,A -85,B 0,C 180,E1 -20200.474,E2 -20200.474} C_VEL
LIN {X 0,Y 220.776,Z 84.986,A -85,B 0,C 180,E1 -20204.454,E2 -20204.454} C_VEL
LIN {X 0,Y 220.772,Z 84.986,A -85,B 0,C 180,E1 -20208.047,E2 -20208.047} C_VEL
LIN {X 0,Y 220.865,Z 85.136,A -85,B 0,C 180,E1 -20211.308,E2 -20211.308} C_VEL
LIN {X 0,Y 223.222,Z 94.912,A -85,B 0,C 180,E1 -20215.478,E2 -20215.478} C_VEL
LIN {X 0,Y 224.142,Z 99.598,A -85,B 0,C 180,E1 -20217.289,E2 -20217.289} C_VEL
LIN {X 0,Y 230.187,Z 115.591,A -85,B 0,C 180,E1 -20218.643,E2 -20218.643} C_VEL
LIN {X 0,Y 233.404,Z 143.471,A -85,B 0,C 180,E1 -20219.982,E2 -20219.982} C_VEL
LIN {X 0,Y 234.805,Z 158.198,A -85,B 0,C 180,E1 -20220.635,E2 -20220.635} C_VEL
LIN {X 0,Y 233.065,Z 209.341,A -85,B 0,C 180,E1 -20222.195,E2 -20222.195} C_VEL
LIN {X 0,Y 231.923,Z 223.191,A -85,B 0,C 180,E1 -20222.964,E2 -20222.964} C_VEL
LIN {X 0,Y 230.421,Z 235.598,A -85,B 0,C 180,E1 -20223.995,E2 -20223.995} C_VEL
LIN {X 0,Y 228.485,Z 248.301,A -85,B 0,C 180,E1 -20225.465,E2 -20225.465} C_VEL
LIN {X 0,Y 226.464,Z 259.609,A -85,B 0,C 180,E1 -20227.174,E2 -20227.174} C_VEL
LIN {X 0,Y 224.8,Z 268.773,A -85,B 0,C 180,E1 -20228.928,E2 -20228.928} C_VEL
LIN {X 0,Y 222.937,Z 277.982,A -85,B 0,C 180,E1 -20231.1,E2 -20231.1} C_VEL
LIN {X 0,Y 221.533,Z 285.881,A -85,B 0,C 180,E1 -20233.41,E2 -20233.41} C_VEL
LIN {X 0,Y 220.201,Z 293.445,A -85,B 0,C 180,E1 -20236.15,E2 -20236.15} C_VEL
LIN {X 0,Y 219.293,Z 299.511,A -85,B 0,C 180,E1 -20238.913,E2 -20238.913} C_VEL
LIN {X 0,Y 218.833,Z 304.3,A -85,B 0,C 180,E1 -20241.69,E2 -20241.69} C_VEL
LIN {X 0,Y 218.723,Z 308.474,A -85,B 0,C 180,E1 -20244.936,E2 -20244.936} C_VEL
LIN {X 0,Y 218.868,Z 311.205,A -85,B 0,C 180,E1 -20248.16,E2 -20248.16} C_VEL
LIN {X 0,Y 218.912,Z 312.178,A -85,B 0,C 180,E1 -20250,E2 -20250} C_VEL
LIN {X 0,Y 218.815,Z 312.744,A -85,B 0,C 180,E1 -20251.84,E2 -20251.84} C_VEL
LIN {X 0,Y 218.701,Z 312.764,A -85,B 0,C 180,E1 -20254.999,E2 -20254.999} C_VEL
LIN {X 0,Y 218.686,Z 311.98,A -85,B 0,C 180,E1 -20257.386,E2 -20257.386} C_VEL
LIN {X 0,Y 219.412,Z 309.514,A -85,B 0,C 180,E1 -20261.08,E2 -20261.08} C_VEL
LIN {X 0,Y 220.445,Z 306.541,A -85,B 0,C 180,E1 -20263.834,E2 -20263.834} C_VEL
LIN {X 0,Y 222.147,Z 302.566,A -85,B 0,C 180,E1 -20266.543,E2 -20266.543} C_VEL
LIN {X 0,Y 224.266,Z 297.479,A -85,B 0,C 180,E1 -20269.211,E2 -20269.211} C_VEL
LIN {X 0,Y 226.693,Z 291.123,A -85,B 0,C 180,E1 -20271.841,E2 -20271.841} C_VEL
LIN {X 0,Y 229.784,Z 283.206,A -85,B 0,C 180,E1 -20274.387,E2 -20274.387} C_VEL
LIN {X 0,Y 233.457,Z 273.389,A -85,B 0,C 180,E1 -20276.844,E2 -20276.844} C_VEL
LIN {X 0,Y 236.866,Z 263.189,A -85,B 0,C 180,E1 -20278.826,E2 -20278.826} C_VEL
LIN {X 0,Y 239.845,Z 253.112,A -85,B 0,C 180,E1 -20280.362,E2 -20280.362} C_VEL
LIN {X 0,Y 242.604,Z 242.153,A -85,B 0,C 180,E1 -20281.673,E2 -20281.673} C_VEL
LIN {X 0,Y 245.184,Z 230.026,A -85,B 0,C 180,E1 -20282.754,E2 -20282.754} C_VEL
LIN {X 0,Y 247.115,Z 216.923,A -85,B 0,C 180,E1 -20283.597,E2 -20283.597} C_VEL
LIN {X 0,Y 248.463,Z 203.403,A -85,B 0,C 180,E1 -20284.124,E2 -20284.124} C_VEL
LIN {X 0,Y 250.248,Z 162.448,A -85,B 0,C 180,E1 -20285.294,E2 -20285.294} C_VEL
LIN {X 0,Y 247.136,Z 140.859,A -85,B 0,C 180,E1 -20286.692,E2 -20286.692} C_VEL
LIN {X 0,Y 240.614,Z 126.274,A -85,B 0,C 180,E1 -20288.612,E2 -20288.612} C_VEL
LIN {X 0,Y 235.31,Z 115.989,A -85,B 0,C 180,E1 -20290.237,E2 -20290.237} C_VEL
LIN {X 0,Y 230.412,Z 107.192,A -85,B 0,C 180,E1 -20291.818,E2 -20291.818} C_VEL
LIN {X 0,Y 227.25,Z 101.961,A -85,B 0,C 180,E1 -20292.881,E2 -20292.881} C_VEL
LIN {X 0,Y 224.644,Z 97.525,A -85,B 0,C 180,E1 -20293.802,E2 -20293.802} C_VEL
LIN {X 0,Y 224.411,Z 97.01,A -85,B 0,C 180,E1 -20293.92,E2 -20293.92} C_VEL
LIN {X 0,Y 222.497,Z 90.484,A -85,B 0,C 180,E1 -20297.697,E2 -20297.697} C_VEL
LIN {X 0,Y 220.787,Z 84.975,A -85,B 0,C 180,E1 -20301.268,E2 -20301.268} C_VEL
LIN {X 0,Y 220.809,Z 84.971,A -85,B 0,C 180,E1 -20305.847,E2 -20305.847} C_VEL
LIN {X 0,Y 220.87,Z 84.965,A -85,B 0,C 180,E1 -20309.395,E2 -20309.395} C_VEL
LIN {X 0,Y 220.898,Z 84.959,A -85,B 0,C 180,E1 -20313.55,E2 -20313.55} C_VEL
LIN {X 0,Y 220.881,Z 84.961,A -85,B 0,C 180,E1 -20317.553,E2 -20317.553} C_VEL
LIN {X 0,Y 220.987,Z 84.944,A -85,B 0,C 180,E1 -20322.571,E2 -20322.571} C_VEL
LIN {X 0,Y 221.015,Z 84.942,A -85,B 0,C 180,E1 -20327.138,E2 -20327.138} C_VEL
LIN {X 0,Y 221.208,Z 84.93,A -85,B 0,C 180,E1 -20330.859,E2 -20330.859} C_VEL
LIN {X 0,Y 221.262,Z 84.907,A -85,B 0,C 180,E1 -20332.7,E2 -20332.7} C_VEL
LIN {X 0,Y 221.514,Z 84.876,A -85,B 0,C 180,E1 -20338.182,E2 -20338.182} C_VEL
LIN {X 0,Y 221.514,Z 84.889,A -85,B 0,C 180,E1 -20341.818,E2 -20341.818} C_VEL
LIN {X 0,Y 221.256,Z 84.919,A -85,B 0,C 180,E1 -20347.299,E2 -20347.299} C_VEL
LIN {X 0,Y 221.068,Z 84.947,A -85,B 0,C 180,E1 -20350.996,E2 -20350.996} C_VEL
LIN {X 0,Y 221.008,Z 84.957,A -85,B 0,C 180,E1 -20356.63,E2 -20356.63} C_VEL
LIN {X 0,Y 220.886,Z 84.97,A -85,B 0,C 180,E1 -20360.487,E2 -20360.487} C_VEL
LIN {X 0,Y 220.853,Z 84.971,A -85,B 0,C 180,E1 -20364.437,E2 -20364.437} C_VEL
LIN {X 0,Y 220.807,Z 84.979,A -85,B 0,C 180,E1 -20368.518,E2 -20368.518} C_VEL
LIN {X 0,Y 220.813,Z 84.979,A -85,B 0,C 180,E1 -20372.757,E2 -20372.757} C_VEL
LIN {X 0,Y 220.827,Z 84.977,A -85,B 0,C 180,E1 -20375.229,E2 -20375.229} C_VEL
LIN {X 0,Y 221.774,Z 87.742,A -85,B 0,C 180,E1 -20375.682,E2 -20375.682} C_VEL
LIN {X 0,Y 223.935,Z 89.977,A -85,B 0,C 180,E1 -20376.424,E2 -20376.424} C_VEL
LIN {X 0,Y 226.442,Z 93.883,A -85,B 0,C 180,E1 -20377.314,E2 -20377.314} C_VEL
LIN {X 0,Y 227.779,Z 95.52,A -85,B 0,C 180,E1 -20377.753,E2 -20377.753} C_VEL
LIN {X 0,Y 234.065,Z 104.655,A -85,B 0,C 180,E1 -20379.769,E2 -20379.769} C_VEL
LIN {X 0,Y 240.842,Z 115.361,A -85,B 0,C 180,E1 -20381.788,E2 -20381.788} C_VEL
LIN {X 0,Y 248.081,Z 127.978,A -85,B 0,C 180,E1 -20383.796,E2 -20383.796} C_VEL
LIN {X 0,Y 251.596,Z 135.566,A -85,B 0,C 180,E1 -20384.763,E2 -20384.763} C_VEL
LIN {X 0,Y 248.938,Z 187.371,A -85,B 0,C 180,E1 -20386.223,E2 -20386.223} C_VEL
LIN {X 0,Y 247.647,Z 200.568,A -85,B 0,C 180,E1 -20386.917,E2 -20386.917} C_VEL
LIN {X 0,Y 245.96,Z 212.811,A -85,B 0,C 180,E1 -20387.881,E2 -20387.881} C_VEL
LIN {X 0,Y 243.809,Z 223.79,A -85,B 0,C 180,E1 -20389.02,E2 -20389.02} C_VEL
LIN {X 0,Y 240.926,Z 235.583,A -85,B 0,C 180,E1 -20390.62,E2 -20390.62} C_VEL
LIN {X 0,Y 237.816,Z 246.457,A -85,B 0,C 180,E1 -20392.525,E2 -20392.525} C_VEL
LIN {X 0,Y 234.433,Z 256.362,A -85,B 0,C 180,E1 -20394.754,E2 -20394.754} C_VEL
LIN {X 0,Y 231.069,Z 265.283,A -85,B 0,C 180,E1 -20397.325,E2 -20397.325} C_VEL
LIN {X 0,Y 228.491,Z 271.521,A -85,B 0,C 180,E1 -20399.612,E2 -20399.612} C_VEL
LIN {X 0,Y 225.958,Z 277.121,A -85,B 0,C 180,E1 -20402.19,E2 -20402.19} C_VEL
LIN {X 0,Y 223.811,Z 281.667,A -85,B 0,C 180,E1 -20404.918,E2 -20404.918} C_VEL
LIN {X 0,Y 222.088,Z 285.084,A -85,B 0,C 180,E1 -20407.682,E2 -20407.682} C_VEL
LIN {X 0,Y 221.117,Z 286.762,A -85,B 0,C 180,E1 -20409.536,E2 -20409.536} C_VEL
LIN {X 0,Y 220.33,Z 288.025,A -85,B 0,C 180,E1 -20411.399,E2 -20411.399} C_VEL
LIN {X 0,Y 219.646,Z 289.009,A -85,B 0,C 180,E1 -20413.721,E2 -20413.721} C_VEL
LIN {X 0,Y 218.96,Z 289.316,A -85,B 0,C 180,E1 -20417.016,E2 -20417.016} C_VEL
LIN {X 0,Y 218.713,Z 288.18,A -85,B 0,C 180,E1 -20420.754,E2 -20420.754} C_VEL
LIN {X 0,Y 219.081,Z 285.844,A -85,B 0,C 180,E1 -20423.968,E2 -20423.968} C_VEL
LIN {X 0,Y 219.413,Z 282.138,A -85,B 0,C 180,E1 -20427.246,E2 -20427.246} C_VEL
LIN {X 0,Y 220.117,Z 277.863,A -85,B 0,C 180,E1 -20430,E2 -20430} C_VEL
LIN {X 0,Y 221.259,Z 271.412,A -85,B 0,C 180,E1 -20433.187,E2 -20433.187} C_VEL
LIN {X 0,Y 222.719,Z 264.325,A -85,B 0,C 180,E1 -20435.887,E2 -20435.887} C_VEL
LIN {X 0,Y 224.432,Z 255.519,A -85,B 0,C 180,E1 -20438.554,E2 -20438.554} C_VEL
LIN {X 0,Y 226.173,Z 246.489,A -85,B 0,C 180,E1 -20440.745,E2 -20440.745} C_VEL
LIN {X 0,Y 228.201,Z 236.457,A -85,B 0,C 180,E1 -20442.676,E2 -20442.676} C_VEL
LIN {X 0,Y 230.012,Z 225.342,A -85,B 0,C 180,E1 -20444.375,E2 -20444.375} C_VEL
LIN {X 0,Y 231.581,Z 212.929,A -85,B 0,C 180,E1 -20445.851,E2 -20445.851} C_VEL
LIN {X 0,Y 232.81,Z 200.233,A -85,B 0,C 180,E1 -20446.948,E2 -20446.948} C_VEL
LIN {X 0,Y 233.681,Z 186.643,A -85,B 0,C 180,E1 -20447.734,E2 -20447.734} C_VEL
LIN {X 0,Y 235.497,Z 135.916,A -85,B 0,C 180,E1 -20449.278,E2 -20449.278} C_VEL
LIN {X 0,Y 235.89,Z 117.953,A -85,B 0,C 180,E1 -20449.831,E2 -20449.831} C_VEL
LIN {X 0,Y 231.555,Z 107.213,A -85,B 0,C 180,E1 -20450.723,E2 -20450.723} C_VEL
LIN {X 0,Y 223.49,Z 90.807,A -85,B 0,C 180,E1 -20452.367,E2 -20452.367} C_VEL
LIN {X 0,Y 221.075,Z 86.003,A -85,B 0,C 180,E1 -20452.884,E2 -20452.884} C_VEL
LIN {X 0,Y 220.875,Z 84.97,A -85,B 0,C 180,E1 -20452.984,E2 -20452.984} C_VEL
LIN {X 0,Y 220.884,Z 84.971,A -85,B 0,C 180,E1 -20457.015,E2 -20457.015} C_VEL
LIN {X 0,Y 220.839,Z 84.973,A -85,B 0,C 180,E1 -20460.768,E2 -20460.768} C_VEL
LIN {X 0,Y 220.817,Z 84.978,A -85,B 0,C 180,E1 -20464.953,E2 -20464.953} C_VEL
LIN {X 0,Y 220.84,Z 84.974,A -85,B 0,C 180,E1 -20467.288,E2 -20467.288} C_VEL
LIN {X 0,Y 220.778,Z 84.982,A -85,B 0,C 180,E1 -20471.951,E2 -20471.951} C_VEL
LIN {X 0,Y 220.772,Z 84.98,A -85,B 0,C 180,E1 -20475.546,E2 -20475.546} C_VEL
LIN {X 0,Y 220.808,Z 84.974,A -85,B 0,C 180,E1 -20480.464,E2 -20480.464} C_VEL
LIN {X 0,Y 220.803,Z 84.976,A -85,B 0,C 180,E1 -20485.046,E2 -20485.046} C_VEL
LIN {X 0,Y 220.87,Z 84.967,A -85,B 0,C 180,E1 -20489.395,E2 -20489.395} C_VEL
LIN {X 0,Y 220.898,Z 84.966,A -85,B 0,C 180,E1 -20493.55,E2 -20493.55} C_VEL
LIN {X 0,Y 220.881,Z 84.97,A -85,B 0,C 180,E1 -20497.554,E2 -20497.554} C_VEL
LIN {X 0,Y 220.988,Z 84.935,A -85,B 0,C 180,E1 -20502.571,E2 -20502.571} C_VEL
LIN {X 0,Y 221.015,Z 84.95,A -85,B 0,C 180,E1 -20507.139,E2 -20507.139} C_VEL
LIN {X 0,Y 221.208,Z 84.927,A -85,B 0,C 180,E1 -20510.86,E2 -20510.86} C_VEL
LIN {X 0,Y 221.262,Z 84.913,A -85,B 0,C 180,E1 -20512.701,E2 -20512.701} C_VEL
LIN {X 0,Y 221.514,Z 84.882,A -85,B 0,C 180,E1 -20518.182,E2 -20518.182} C_VEL
LIN {X 0,Y 221.514,Z 84.893,A -85,B 0,C 180,E1 -20521.818,E2 -20521.818} C_VEL
LIN {X 0,Y 221.25,Z 84.925,A -85,B 0,C 180,E1 -20527.3,E2 -20527.3} C_VEL
LIN {X 0,Y 221.066,Z 84.943,A -85,B 0,C 180,E1 -20530.997,E2 -20530.997} C_VEL
LIN {X 0,Y 221.01,Z 84.952,A -85,B 0,C 180,E1 -20536.631,E2 -20536.631} C_VEL
LIN {X 0,Y 220.888,Z 84.966,A -85,B 0,C 180,E1 -20540.487,E2 -20540.487} C_VEL
LIN {X 0,Y 220.854,Z 84.974,A -85,B 0,C 180,E1 -20544.437,E2 -20544.437} C_VEL
LIN {X 0,Y 220.809,Z 84.982,A -85,B 0,C 180,E1 -20548.518,E2 -20548.518} C_VEL
LIN {X 0,Y 220.815,Z 84.982,A -85,B 0,C 180,E1 -20552.757,E2 -20552.757} C_VEL
LIN {X 0,Y 220.813,Z 84.98,A -85,B 0,C 180,E1 -20557.278,E2 -20557.278} C_VEL
LIN {X 0,Y 220.78,Z 84.983,A -85,B 0,C 180,E1 -20560.474,E2 -20560.474} C_VEL
LIN {X 0,Y 220.044,Z 85.077,A -85,B 0,C 180,E1 -20561.994,E2 -20561.994} C_VEL
LIN {X 0,Y 217.124,Z 85.441,A -85,B 0,C 180,E1 -20564.475,E2 -20564.475} C_VEL
LIN {X 0,Y 214.715,Z 85.741,A -85,B 0,C 180,E1 -20566.501,E2 -20566.501} C_VEL
LIN {X 0,Y 213.743,Z 85.861,A -85,B 0,C 180,E1 -20568.076,E2 -20568.076} C_VEL
LIN {X 0,Y 213.694,Z 85.867,A -85,B 0,C 180,E1 -20568.609,E2 -20568.609} C_VEL
LIN {X 0,Y 213.78,Z 85.867,A -85,B 0,C 180,E1 -20570.486,E2 -20570.486} C_VEL
LIN {X 0,Y 215.927,Z 94.779,A -85,B 0,C 180,E1 -20574.46,E2 -20574.46} C_VEL
LIN {X 0,Y 216.883,Z 99.186,A -85,B 0,C 180,E1 -20576.243,E2 -20576.243} C_VEL
LIN {X 0,Y 223.989,Z 117.453,A -85,B 0,C 180,E1 -20577.905,E2 -20577.905} C_VEL
LIN {X 0,Y 227.006,Z 144.157,A -85,B 0,C 180,E1 -20579.232,E2 -20579.232} C_VEL
LIN {X 0,Y 228.345,Z 159.528,A -85,B 0,C 180,E1 -20579.927,E2 -20579.927} C_VEL
LIN {X 0,Y 226.606,Z 208.265,A -85,B 0,C 180,E1 -20581.44,E2 -20581.44} C_VEL
LIN {X 0,Y 225.509,Z 221.795,A -85,B 0,C 180,E1 -20582.192,E2 -20582.192} C_VEL
LIN {X 0,Y 224.063,Z 233.948,A -85,B 0,C 180,E1 -20583.199,E2 -20583.199} C_VEL
LIN {X 0,Y 222.35,Z 245.403,A -85,B 0,C 180,E1 -20584.49,E2 -20584.49} C_VEL
LIN {X 0,Y 220.099,Z 257.156,A -85,B 0,C 180,E1 -20586.226,E2 -20586.226} C_VEL
LIN {X 0,Y 218.132,Z 267.761,A -85,B 0,C 180,E1 -20588.252,E2 -20588.252} C_VEL
LIN {X 0,Y 216.23,Z 277.115,A -85,B 0,C 180,E1 -20590.489,E2 -20590.489} C_VEL
LIN {X 0,Y 215.385,Z 281.023,A -85,B 0,C 180,E1 -20591.585,E2 -20591.585} C_VEL
LIN {X 0,Y 213.956,Z 289.125,A -85,B 0,C 180,E1 -20594.276,E2 -20594.276} C_VEL
LIN {X 0,Y 212.675,Z 295.964,A -85,B 0,C 180,E1 -20597.111,E2 -20597.111} C_VEL
LIN {X 0,Y 211.907,Z 302.249,A -85,B 0,C 180,E1 -20600.454,E2 -20600.454} C_VEL
LIN {X 0,Y 211.641,Z 306.317,A -85,B 0,C 180,E1 -20603.326,E2 -20603.326} C_VEL
LIN {X 0,Y 211.667,Z 309.309,A -85,B 0,C 180,E1 -20606.192,E2 -20606.192} C_VEL
LIN {X 0,Y 211.795,Z 310.74,A -85,B 0,C 180,E1 -20608.098,E2 -20608.098} C_VEL
LIN {X 0,Y 211.84,Z 311.737,A -85,B 0,C 180,E1 -20610,E2 -20610} C_VEL
LIN {X 0,Y 211.743,Z 312.325,A -85,B 0,C 180,E1 -20611.902,E2 -20611.902} C_VEL
LIN {X 0,Y 211.606,Z 312.422,A -85,B 0,C 180,E1 -20614.873,E2 -20614.873} C_VEL
LIN {X 0,Y 211.625,Z 311.651,A -85,B 0,C 180,E1 -20617.634,E2 -20617.634} C_VEL
LIN {X 0,Y 212.402,Z 309.233,A -85,B 0,C 180,E1 -20621.451,E2 -20621.451} C_VEL
LIN {X 0,Y 213.515,Z 306.308,A -85,B 0,C 180,E1 -20624.292,E2 -20624.292} C_VEL
LIN {X 0,Y 215.317,Z 302.384,A -85,B 0,C 180,E1 -20627.083,E2 -20627.083} C_VEL
LIN {X 0,Y 217.557,Z 297.354,A -85,B 0,C 180,E1 -20629.828,E2 -20629.828} C_VEL
LIN {X 0,Y 220.082,Z 291.067,A -85,B 0,C 180,E1 -20632.532,E2 -20632.532} C_VEL
LIN {X 0,Y 223.338,Z 283.251,A -85,B 0,C 180,E1 -20635.139,E2 -20635.139} C_VEL
LIN {X 0,Y 227.16,Z 273.523,A -85,B 0,C 180,E1 -20637.651,E2 -20637.651} C_VEL
LIN {X 0,Y 230.69,Z 263.485,A -85,B 0,C 180,E1 -20639.674,E2 -20639.674} C_VEL
LIN {X 0,Y 233.771,Z 253.565,A -85,B 0,C 180,E1 -20641.238,E2 -20641.238} C_VEL
LIN {X 0,Y 236.612,Z 242.812,A -85,B 0,C 180,E1 -20642.572,E2 -20642.572} C_VEL
LIN {X 0,Y 239.499,Z 229.853,A -85,B 0,C 180,E1 -20643.76,E2 -20643.76} C_VEL
LIN {X 0,Y 241.462,Z 217.203,A -85,B 0,C 180,E1 -20644.597,E2 -20644.597} C_VEL
LIN {X 0,Y 242.845,Z 204.531,A -85,B 0,C 180,E1 -20645.113,E2 -20645.113} C_VEL
LIN {X 0,Y 244.741,Z 163.589,A -85,B 0,C 180,E1 -20646.308,E2 -20646.308} C_VEL
LIN {X 0,Y 241.998,Z 144.011,A -85,B 0,C 180,E1 -20647.617,E2 -20647.617} C_VEL
LIN {X 0,Y 236.014,Z 130.356,A -85,B 0,C 180,E1 -20649.475,E2 -20649.475} C_VEL
LIN {X 0,Y 230.821,Z 120.081,A -85,B 0,C 180,E1 -20651.152,E2 -20651.152} C_VEL
LIN {X 0,Y 226.215,Z 111.773,A -85,B 0,C 180,E1 -20652.713,E2 -20652.713} C_VEL
LIN {X 0,Y 223.061,Z 106.483,A -85,B 0,C 180,E1 -20653.828,E2 -20653.828} C_VEL
LIN {X 0,Y 219.905,Z 101.278,A -85,B 0,C 180,E1 -20655,E2 -20655} C_VEL
LIN {X 0,Y 217.255,Z 96.977,A -85,B 0,C 180,E1 -20656.03,E2 -20656.03} C_VEL
LIN {X 0,Y 216.996,Z 96.336,A -85,B 0,C 180,E1 -20656.202,E2 -20656.202} C_VEL
LIN {X 0,Y 214.956,Z 89.742,A -85,B 0,C 180,E1 -20660.39,E2 -20660.39} C_VEL
LIN {X 0,Y 213.756,Z 85.846,A -85,B 0,C 180,E1 -20663.144,E2 -20663.144} C_VEL
LIN {X 0,Y 213.759,Z 85.848,A -85,B 0,C 180,E1 -20666.018,E2 -20666.018} C_VEL
LIN {X 0,Y 213.783,Z 85.845,A -85,B 0,C 180,E1 -20670.454,E2 -20670.454} C_VEL
LIN {X 0,Y 213.804,Z 85.843,A -85,B 0,C 180,E1 -20674.702,E2 -20674.702} C_VEL
LIN {X 0,Y 213.815,Z 85.839,A -85,B 0,C 180,E1 -20678.803,E2 -20678.803} C_VEL
LIN {X 0,Y 213.947,Z 85.82,A -85,B 0,C 180,E1 -20682.804,E2 -20682.804} C_VEL
LIN {X 0,Y 213.956,Z 85.824,A -85,B 0,C 180,E1 -20686.707,E2 -20686.707} C_VEL
LIN {X 0,Y 214.145,Z 85.811,A -85,B 0,C 180,E1 -20690.555,E2 -20690.555} C_VEL
LIN {X 0,Y 214.102,Z 85.804,A -85,B 0,C 180,E1 -20694.348,E2 -20694.348} C_VEL
LIN {X 0,Y 214.447,Z 85.756,A -85,B 0,C 180,E1 -20698.122,E2 -20698.122} C_VEL
LIN {X 0,Y 214.553,Z 85.753,A -85,B 0,C 180,E1 -20700,E2 -20700} C_VEL
LIN {X 0,Y 214.447,Z 85.769,A -85,B 0,C 180,E1 -20701.878,E2 -20701.878} C_VEL
LIN {X 0,Y 214.196,Z 85.796,A -85,B 0,C 180,E1 -20707.541,E2 -20707.541} C_VEL
LIN {X 0,Y 213.999,Z 85.83,A -85,B 0,C 180,E1 -20711.364,E2 -20711.364} C_VEL
LIN {X 0,Y 213.922,Z 85.83,A -85,B 0,C 180,E1 -20715.238,E2 -20715.238} C_VEL
LIN {X 0,Y 213.835,Z 85.837,A -85,B 0,C 180,E1 -20719.188,E2 -20719.188} C_VEL
LIN {X 0,Y 213.806,Z 85.841,A -85,B 0,C 180,E1 -20723.232,E2 -20723.232} C_VEL
LIN {X 0,Y 213.789,Z 85.845,A -85,B 0,C 180,E1 -20727.428,E2 -20727.428} C_VEL
LIN {X 0,Y 213.759,Z 85.854,A -85,B 0,C 180,E1 -20731.739,E2 -20731.739} C_VEL
LIN {X 0,Y 213.769,Z 85.854,A -85,B 0,C 180,E1 -20732.992,E2 -20732.992} C_VEL
LIN {X 0,Y 214.764,Z 88.713,A -85,B 0,C 180,E1 -20733.519,E2 -20733.519} C_VEL
LIN {X 0,Y 216.86,Z 90.878,A -85,B 0,C 180,E1 -20734.318,E2 -20734.318} C_VEL
LIN {X 0,Y 217.537,Z 91.697,A -85,B 0,C 180,E1 -20734.576,E2 -20734.576} C_VEL
LIN {X 0,Y 219.729,Z 94.976,A -85,B 0,C 180,E1 -20735.421,E2 -20735.421} C_VEL
LIN {X 0,Y 221.09,Z 96.643,A -85,B 0,C 180,E1 -20735.912,E2 -20735.912} C_VEL
LIN {X 0,Y 223.535,Z 100.032,A -85,B 0,C 180,E1 -20736.787,E2 -20736.787} C_VEL
LIN {X 0,Y 230.066,Z 109.596,A -85,B 0,C 180,E1 -20738.983,E2 -20738.983} C_VEL
LIN {X 0,Y 237.809,Z 122.032,A -85,B 0,C 180,E1 -20741.378,E2 -20741.378} C_VEL
LIN {X 0,Y 244.163,Z 133.63,A -85,B 0,C 180,E1 -20743.215,E2 -20743.215} C_VEL
LIN {X 0,Y 246.083,Z 137.813,A -85,B 0,C 180,E1 -20743.767,E2 -20743.767} C_VEL
LIN {X 0,Y 243.421,Z 187.511,A -85,B 0,C 180,E1 -20745.186,E2 -20745.186} C_VEL
LIN {X 0,Y 242.064,Z 200.888,A -85,B 0,C 180,E1 -20745.897,E2 -20745.897} C_VEL
LIN {X 0,Y 240.343,Z 212.841,A -85,B 0,C 180,E1 -20746.845,E2 -20746.845} C_VEL
LIN {X 0,Y 237.978,Z 224.485,A -85,B 0,C 180,E1 -20748.074,E2 -20748.074} C_VEL
LIN {X 0,Y 234.978,Z 236.221,A -85,B 0,C 180,E1 -20749.7,E2 -20749.7} C_VEL
LIN {X 0,Y 231.832,Z 246.728,A -85,B 0,C 180,E1 -20751.577,E2 -20751.577} C_VEL
LIN {X 0,Y 228.491,Z 256.184,A -85,B 0,C 180,E1 -20753.729,E2 -20753.729} C_VEL
LIN {X 0,Y 224.949,Z 265.108,A -85,B 0,C 180,E1 -20756.32,E2 -20756.32} C_VEL
LIN {X 0,Y 221.986,Z 272.025,A -85,B 0,C 180,E1 -20758.896,E2 -20758.896} C_VEL
LIN {X 0,Y 219.541,Z 277.141,A -85,B 0,C 180,E1 -20761.303,E2 -20761.303} C_VEL
LIN {X 0,Y 217.222,Z 281.781,A -85,B 0,C 180,E1 -20764.101,E2 -20764.101} C_VEL
LIN {X 0,Y 215.384,Z 285.272,A -85,B 0,C 180,E1 -20766.948,E2 -20766.948} C_VEL
LIN {X 0,Y 214.314,Z 287.002,A -85,B 0,C 180,E1 -20768.855,E2 -20768.855} C_VEL
LIN {X 0,Y 212.828,Z 289.192,A -85,B 0,C 180,E1 -20772.711,E2 -20772.711} C_VEL
LIN {X 0,Y 212.315,Z 289.675,A -85,B 0,C 180,E1 -20774.644,E2 -20774.644} C_VEL
LIN {X 0,Y 211.686,Z 289.383,A -85,B 0,C 180,E1 -20778.51,E2 -20778.51} C_VEL
LIN {X 0,Y 211.637,Z 288.654,A -85,B 0,C 180,E1 -20780.442,E2 -20780.442} C_VEL
LIN {X 0,Y 211.996,Z 286.181,A -85,B 0,C 180,E1 -20784.013,E2 -20784.013} C_VEL
LIN {X 0,Y 212.316,Z 282.777,A -85,B 0,C 180,E1 -20787.154,E2 -20787.154} C_VEL
LIN {X 0,Y 213.024,Z 278.577,A -85,B 0,C 180,E1 -20790,E2 -20790} C_VEL
LIN {X 0,Y 214.154,Z 272.215,A -85,B 0,C 180,E1 -20793.293,E2 -20793.293} C_VEL
LIN {X 0,Y 215.672,Z 265.261,A -85,B 0,C 180,E1 -20796.08,E2 -20796.08} C_VEL
LIN {X 0,Y 217.43,Z 256.57,A -85,B 0,C 180,E1 -20798.832,E2 -20798.832} C_VEL
LIN {X 0,Y 219.241,Z 247.669,A -85,B 0,C 180,E1 -20801.089,E2 -20801.089} C_VEL
LIN {X 0,Y 221.333,Z 237.839,A -85,B 0,C 180,E1 -20803.076,E2 -20803.076} C_VEL
LIN {X 0,Y 223.211,Z 227.013,A -85,B 0,C 180,E1 -20804.823,E2 -20804.823} C_VEL
LIN {X 0,Y 224.862,Z 214.921,A -85,B 0,C 180,E1 -20806.338,E2 -20806.338} C_VEL
LIN {X 0,Y 226.169,Z 202.282,A -85,B 0,C 180,E1 -20807.52,E2 -20807.52} C_VEL
LIN {X 0,Y 227.09,Z 189.389,A -85,B 0,C 180,E1 -20808.336,E2 -20808.336} C_VEL
LIN {X 0,Y 227.813,Z 171.418,A -85,B 0,C 180,E1 -20808.979,E2 -20808.979} C_VEL
LIN {X 0,Y 229.581,Z 119.779,A -85,B 0,C 180,E1 -20810.539,E2 -20810.539} C_VEL
LIN {X 0,Y 223.94,Z 106.505,A -85,B 0,C 180,E1 -20811.742,E2 -20811.742} C_VEL
LIN {X 0,Y 216.661,Z 92.07,A -85,B 0,C 180,E1 -20813.307,E2 -20813.307} C_VEL
LIN {X 0,Y 214.052,Z 86.954,A -85,B 0,C 180,E1 -20813.896,E2 -20813.896} C_VEL
LIN {X 0,Y 213.841,Z 85.846,A -85,B 0,C 180,E1 -20813.992,E2 -20813.992} C_VEL
LIN {X 0,Y 213.83,Z 85.85,A -85,B 0,C 180,E1 -20817.45,E2 -20817.45} C_VEL
LIN {X 0,Y 213.771,Z 85.855,A -85,B 0,C 180,E1 -20821.737,E2 -20821.737} C_VEL
LIN {X 0,Y 213.754,Z 85.858,A -85,B 0,C 180,E1 -20826.287,E2 -20826.287} C_VEL
LIN {X 0,Y 213.719,Z 85.859,A -85,B 0,C 180,E1 -20831.124,E2 -20831.124} C_VEL
LIN {X 0,Y 213.708,Z 85.863,A -85,B 0,C 180,E1 -20833.679,E2 -20833.679} C_VEL
LIN {X 0,Y 213.704,Z 85.861,A -85,B 0,C 180,E1 -20836.345,E2 -20836.345} C_VEL
LIN {X 0,Y 213.718,Z 85.859,A -85,B 0,C 180,E1 -20839.144,E2 -20839.144} C_VEL
LIN {X 0,Y 213.745,Z 85.854,A -85,B 0,C 180,E1 -20843.712,E2 -20843.712} C_VEL
LIN {X 0,Y 213.797,Z 85.85,A -85,B 0,C 180,E1 -20848.725,E2 -20848.725} C_VEL
LIN {X 0,Y 213.828,Z 85.85,A -85,B 0,C 180,E1 -20852.604,E2 -20852.604} C_VEL
LIN {X 0,Y 213.855,Z 85.847,A -85,B 0,C 180,E1 -20856.953,E2 -20856.953} C_VEL
LIN {X 0,Y 213.947,Z 85.81,A -85,B 0,C 180,E1 -20862.804,E2 -20862.804} C_VEL
LIN {X 0,Y 213.956,Z 85.826,A -85,B 0,C 180,E1 -20866.707,E2 -20866.707} C_VEL
LIN {X 0,Y 214.145,Z 85.808,A -85,B 0,C 180,E1 -20870.556,E2 -20870.556} C_VEL
LIN {X 0,Y 214.1,Z 85.792,A -85,B 0,C 180,E1 -20874.349,E2 -20874.349} C_VEL
LIN {X 0,Y 214.447,Z 85.761,A -85,B 0,C 180,E1 -20878.122,E2 -20878.122} C_VEL
LIN {X 0,Y 214.554,Z 85.758,A -85,B 0,C 180,E1 -20880,E2 -20880} C_VEL
LIN {X 0,Y 214.447,Z 85.773,A -85,B 0,C 180,E1 -20881.878,E2 -20881.878} C_VEL
LIN {X 0,Y 214.191,Z 85.806,A -85,B 0,C 180,E1 -20887.542,E2 -20887.542} C_VEL
LIN {X 0,Y 213.997,Z 85.825,A -85,B 0,C 180,E1 -20891.365,E2 -20891.365} C_VEL
LIN {X 0,Y 213.92,Z 85.835,A -85,B 0,C 180,E1 -20895.238,E2 -20895.238} C_VEL
LIN {X 0,Y 213.837,Z 85.848,A -85,B 0,C 180,E1 -20899.188,E2 -20899.188} C_VEL
LIN {X 0,Y 213.807,Z 85.854,A -85,B 0,C 180,E1 -20903.232,E2 -20903.232} C_VEL
LIN {X 0,Y 213.791,Z 85.856,A -85,B 0,C 180,E1 -20907.429,E2 -20907.429} C_VEL
LIN {X 0,Y 213.761,Z 85.859,A -85,B 0,C 180,E1 -20911.739,E2 -20911.739} C_VEL
LIN {X 0,Y 213.747,Z 85.862,A -85,B 0,C 180,E1 -20916.288,E2 -20916.288} C_VEL
LIN {X 0,Y 213.715,Z 85.864,A -85,B 0,C 180,E1 -20921.125,E2 -20921.125} C_VEL
LIN {X 0,Y 213.709,Z 85.863,A -85,B 0,C 180,E1 -20923.678,E2 -20923.678} C_VEL
LIN {X 0,Y 213.709,Z 85.866,A -85,B 0,C 180,E1 -20926.344,E2 -20926.344} C_VEL
LIN {X 0,Y 213.694,Z 85.867,A -85,B 0,C 180,E1 -20928.609,E2 -20928.609} C_VEL
LIN {X 0,Y 213.184,Z 86.46,A -85,B 0,C 180,E1 -20929.644,E2 -20929.644} C_VEL
LIN {X 0,Y 211.943,Z 87.907,A -85,B 0,C 180,E1 -20930.599,E2 -20930.599} C_VEL
LIN {X 0,Y 208.926,Z 92.946,A -85,B 0,C 180,E1 -20932.685,E2 -20932.685} C_VEL
LIN {X 0,Y 208.764,Z 95.217,A -85,B 0,C 180,E1 -20933.626,E2 -20933.626} C_VEL
LIN {X 0,Y 209.561,Z 98.57,A -85,B 0,C 180,E1 -20935.098,E2 -20935.098} C_VEL
LIN {X 0,Y 217.829,Z 119.516,A -85,B 0,C 180,E1 -20937.134,E2 -20937.134} C_VEL
LIN {X 0,Y 220.662,Z 144.988,A -85,B 0,C 180,E1 -20938.449,E2 -20938.449} C_VEL
LIN {X 0,Y 221.953,Z 159.719,A -85,B 0,C 180,E1 -20939.143,E2 -20939.143} C_VEL
LIN {X 0,Y 220.119,Z 208.687,A -85,B 0,C 180,E1 -20940.715,E2 -20940.715} C_VEL
LIN {X 0,Y 218.983,Z 221.936,A -85,B 0,C 180,E1 -20941.484,E2 -20941.484} C_VEL
LIN {X 0,Y 217.41,Z 234.507,A -85,B 0,C 180,E1 -20942.571,E2 -20942.571} C_VEL
LIN {X 0,Y 215.64,Z 245.697,A -85,B 0,C 180,E1 -20943.897,E2 -20943.897} C_VEL
LIN {X 0,Y 213.314,Z 257.32,A -85,B 0,C 180,E1 -20945.68,E2 -20945.68} C_VEL
LIN {X 0,Y 211.285,Z 267.833,A -85,B 0,C 180,E1 -20947.767,E2 -20947.767} C_VEL
LIN {X 0,Y 209.347,Z 277.003,A -85,B 0,C 180,E1 -20950.051,E2 -20950.051} C_VEL
LIN {X 0,Y 208.53,Z 279.88,A -85,B 0,C 180,E1 -20950.87,E2 -20950.87} C_VEL
LIN {X 0,Y 207.564,Z 285.691,A -85,B 0,C 180,E1 -20952.766,E2 -20952.766} C_VEL
LIN {X 0,Y 206.13,Z 293.153,A -85,B 0,C 180,E1 -20955.688,E2 -20955.688} C_VEL
LIN {X 0,Y 205.046,Z 299.992,A -85,B 0,C 180,E1 -20959.134,E2 -20959.134} C_VEL
LIN {X 0,Y 204.619,Z 304.494,A -85,B 0,C 180,E1 -20962.103,E2 -20962.103} C_VEL
LIN {X 0,Y 204.559,Z 307.925,A -85,B 0,C 180,E1 -20965.107,E2 -20965.107} C_VEL
LIN {X 0,Y 204.699,Z 310.274,A -85,B 0,C 180,E1 -20968.032,E2 -20968.032} C_VEL
LIN {X 0,Y 204.769,Z 311.296,A -85,B 0,C 180,E1 -20970,E2 -20970} C_VEL
LIN {X 0,Y 204.672,Z 311.907,A -85,B 0,C 180,E1 -20971.968,E2 -20971.968} C_VEL
LIN {X 0,Y 204.539,Z 312.072,A -85,B 0,C 180,E1 -20974.829,E2 -20974.829} C_VEL
LIN {X 0,Y 204.582,Z 311.323,A -85,B 0,C 180,E1 -20977.898,E2 -20977.898} C_VEL
LIN {X 0,Y 205.412,Z 308.95,A -85,B 0,C 180,E1 -20981.846,E2 -20981.846} C_VEL
LIN {X 0,Y 206.612,Z 306.075,A -85,B 0,C 180,E1 -20984.78,E2 -20984.78} C_VEL
LIN {X 0,Y 208.492,Z 302.205,A -85,B 0,C 180,E1 -20987.661,E2 -20987.661} C_VEL
LIN {X 0,Y 210.853,Z 297.233,A -85,B 0,C 180,E1 -20990.486,E2 -20990.486} C_VEL
LIN {X 0,Y 213.512,Z 291.011,A -85,B 0,C 180,E1 -20993.266,E2 -20993.266} C_VEL
LIN {X 0,Y 216.918,Z 283.305,A -85,B 0,C 180,E1 -20995.938,E2 -20995.938} C_VEL
LIN {X 0,Y 220.902,Z 273.665,A -85,B 0,C 180,E1 -20998.504,E2 -20998.504} C_VEL
LIN {X 0,Y 224.564,Z 263.748,A -85,B 0,C 180,E1 -21000.568,E2 -21000.568} C_VEL
LIN {X 0,Y 227.757,Z 254.006,A -85,B 0,C 180,E1 -21002.16,E2 -21002.16} C_VEL
LIN {X 0,Y 230.684,Z 243.473,A -85,B 0,C 180,E1 -21003.518,E2 -21003.518} C_VEL
LIN {X 0,Y 233.637,Z 230.81,A -85,B 0,C 180,E1 -21004.726,E2 -21004.726} C_VEL
LIN {X 0,Y 235.79,Z 218.113,A -85,B 0,C 180,E1 -21005.608,E2 -21005.608} C_VEL
LIN {X 0,Y 237.291,Z 205.552,A -85,B 0,C 180,E1 -21006.156,E2 -21006.156} C_VEL
LIN {X 0,Y 239.305,Z 164.859,A -85,B 0,C 180,E1 -21007.365,E2 -21007.365} C_VEL
LIN {X 0,Y 236.919,Z 147.007,A -85,B 0,C 180,E1 -21008.591,E2 -21008.591} C_VEL
LIN {X 0,Y 231.173,Z 133.851,A -85,B 0,C 180,E1 -21010.472,E2 -21010.472} C_VEL
LIN {X 0,Y 225.336,Z 122.035,A -85,B 0,C 180,E1 -21012.481,E2 -21012.481} C_VEL
LIN {X 0,Y 219.233,Z 111.436,A -85,B 0,C 180,E1 -21014.703,E2 -21014.703} C_VEL
LIN {X 0,Y 216.056,Z 106.191,A -85,B 0,C 180,E1 -21015.94,E2 -21015.94} C_VEL
LIN {X 0,Y 212.872,Z 101.097,A -85,B 0,C 180,E1 -21017.244,E2 -21017.244} C_VEL
LIN {X 0,Y 209.901,Z 96.529,A -85,B 0,C 180,E1 -21018.522,E2 -21018.522} C_VEL
LIN {X 0,Y 209.502,Z 95.575,A -85,B 0,C 180,E1 -21018.826,E2 -21018.826} C_VEL
LIN {X 0,Y 207.817,Z 90.33,A -85,B 0,C 180,E1 -21022.502,E2 -21022.502} C_VEL
LIN {X 0,Y 206.737,Z 86.727,A -85,B 0,C 180,E1 -21025.29,E2 -21025.29} C_VEL
LIN {X 0,Y 206.725,Z 86.727,A -85,B 0,C 180,E1 -21029.339,E2 -21029.339} C_VEL
LIN {X 0,Y 206.735,Z 86.722,A -85,B 0,C 180,E1 -21033.772,E2 -21033.772} C_VEL
LIN {X 0,Y 206.76,Z 86.717,A -85,B 0,C 180,E1 -21038.043,E2 -21038.043} C_VEL
LIN {X 0,Y 206.879,Z 86.703,A -85,B 0,C 180,E1 -21042.197,E2 -21042.197} C_VEL
LIN {X 0,Y 206.899,Z 86.708,A -85,B 0,C 180,E1 -21046.244,E2 -21046.244} C_VEL
LIN {X 0,Y 207.102,Z 86.688,A -85,B 0,C 180,E1 -21050.231,E2 -21050.231} C_VEL
LIN {X 0,Y 207.063,Z 86.679,A -85,B 0,C 180,E1 -21054.156,E2 -21054.156} C_VEL
LIN {X 0,Y 207.384,Z 86.636,A -85,B 0,C 180,E1 -21058.058,E2 -21058.058} C_VEL
LIN {X 0,Y 207.518,Z 86.629,A -85,B 0,C 180,E1 -21060,E2 -21060} C_VEL
LIN {X 0,Y 207.383,Z 86.648,A -85,B 0,C 180,E1 -21061.942,E2 -21061.942} C_VEL
LIN {X 0,Y 207.139,Z 86.672,A -85,B 0,C 180,E1 -21067.8,E2 -21067.8} C_VEL
LIN {X 0,Y 206.923,Z 86.71,A -85,B 0,C 180,E1 -21071.758,E2 -21071.758} C_VEL
LIN {X 0,Y 206.858,Z 86.715,A -85,B 0,C 180,E1 -21075.771,E2 -21075.771} C_VEL
LIN {X 0,Y 206.764,Z 86.722,A -85,B 0,C 180,E1 -21079.871,E2 -21079.871} C_VEL
LIN {X 0,Y 206.741,Z 86.725,A -85,B 0,C 180,E1 -21084.075,E2 -21084.075} C_VEL
LIN {X 0,Y 206.719,Z 86.732,A -85,B 0,C 180,E1 -21088.422,E2 -21088.422} C_VEL
LIN {X 0,Y 206.713,Z 86.74,A -85,B 0,C 180,E1 -21090.521,E2 -21090.521} C_VEL
LIN {X 0,Y 207.473,Z 89.162,A -85,B 0,C 180,E1 -21090.953,E2 -21090.953} C_VEL
LIN {X 0,Y 209.553,Z 91.565,A -85,B 0,C 180,E1 -21091.862,E2 -21091.862} C_VEL
LIN {X 0,Y 210.571,Z 92.446,A -85,B 0,C 180,E1 -21092.277,E2 -21092.277} C_VEL
LIN {X 0,Y 212.538,Z 95.634,A -85,B 0,C 180,E1 -21093.137,E2 -21093.137} C_VEL
LIN {X 0,Y 214.391,Z 97.688,A -85,B 0,C 180,E1 -21093.868,E2 -21093.868} C_VEL
LIN {X 0,Y 217.048,Z 101.263,A -85,B 0,C 180,E1 -21094.906,E2 -21094.906} C_VEL
LIN {X 0,Y 224.174,Z 111.615,A -85,B 0,C 180,E1 -21097.509,E2 -21097.509} C_VEL
LIN {X 0,Y 230.604,Z 121.74,A -85,B 0,C 180,E1 -21099.65,E2 -21099.65} C_VEL
LIN {X 0,Y 238.283,Z 135.193,A -85,B 0,C 180,E1 -21102.019,E2 -21102.019} C_VEL
LIN {X 0,Y 240.64,Z 140.223,A -85,B 0,C 180,E1 -21102.732,E2 -21102.732} C_VEL
LIN {X 0,Y 237.995,Z 187.579,A -85,B 0,C 180,E1 -21104.099,E2 -21104.099} C_VEL
LIN {X 0,Y 236.684,Z 200.361,A -85,B 0,C 180,E1 -21104.776,E2 -21104.776} C_VEL
LIN {X 0,Y 234.778,Z 213.15,A -85,B 0,C 180,E1 -21105.79,E2 -21105.79} C_VEL
LIN {X 0,Y 232.221,Z 225.18,A -85,B 0,C 180,E1 -21107.082,E2 -21107.082} C_VEL
LIN {X 0,Y 229.097,Z 236.858,A -85,B 0,C 180,E1 -21108.734,E2 -21108.734} C_VEL
LIN {X 0,Y 225.818,Z 247.313,A -85,B 0,C 180,E1 -21110.645,E2 -21110.645} C_VEL
LIN {X 0,Y 222.586,Z 256.095,A -85,B 0,C 180,E1 -21112.672,E2 -21112.672} C_VEL
LIN {X 0,Y 218.915,Z 264.939,A -85,B 0,C 180,E1 -21115.261,E2 -21115.261} C_VEL
LIN {X 0,Y 215.864,Z 271.798,A -85,B 0,C 180,E1 -21117.832,E2 -21117.832} C_VEL
LIN {X 0,Y 213.171,Z 277.159,A -85,B 0,C 180,E1 -21120.361,E2 -21120.361} C_VEL
LIN {X 0,Y 210.686,Z 281.88,A -85,B 0,C 180,E1 -21123.235,E2 -21123.235} C_VEL
LIN {X 0,Y 208.682,Z 285.444,A -85,B 0,C 180,E1 -21126.163,E2 -21126.163} C_VEL
LIN {X 0,Y 207.546,Z 287.243,A -85,B 0,C 180,E1 -21128.131,E2 -21128.131} C_VEL
LIN {X 0,Y 205.918,Z 289.5,A -85,B 0,C 180,E1 -21132.111,E2 -21132.111} C_VEL
LIN {X 0,Y 205.366,Z 290.032,A -85,B 0,C 180,E1 -21134.111,E2 -21134.111} C_VEL
LIN {X 0,Y 204.918,Z 290.129,A -85,B 0,C 180,E1 -21136.109,E2 -21136.109} C_VEL
LIN {X 0,Y 204.546,Z 289.126,A -85,B 0,C 180,E1 -21140.108,E2 -21140.108} C_VEL
LIN {X 0,Y 204.614,Z 288.037,A -85,B 0,C 180,E1 -21142.103,E2 -21142.103} C_VEL
LIN {X 0,Y 204.919,Z 286.487,A -85,B 0,C 180,E1 -21144.095,E2 -21144.095} C_VEL
LIN {X 0,Y 205.223,Z 283.416,A -85,B 0,C 180,E1 -21147.056,E2 -21147.056} C_VEL
LIN {X 0,Y 205.934,Z 279.292,A -85,B 0,C 180,E1 -21150,E2 -21150} C_VEL
LIN {X 0,Y 207.059,Z 273.014,A -85,B 0,C 180,E1 -21153.405,E2 -21153.405} C_VEL
LIN {X 0,Y 208.632,Z 266.163,A -85,B 0,C 180,E1 -21156.286,E2 -21156.286} C_VEL
LIN {X 0,Y 210.439,Z 257.619,A -85,B 0,C 180,E1 -21159.128,E2 -21159.128} C_VEL
LIN {X 0,Y 212.322,Z 248.846,A -85,B 0,C 180,E1 -21161.456,E2 -21161.456} C_VEL
LIN {X 0,Y 214.479,Z 239.175,A -85,B 0,C 180,E1 -21163.502,E2 -21163.502} C_VEL
LIN {X 0,Y 216.424,Z 228.626,A -85,B 0,C 180,E1 -21165.299,E2 -21165.299} C_VEL
LIN {X 0,Y 218.15,Z 216.903,A -85,B 0,C 180,E1 -21166.855,E2 -21166.855} C_VEL
LIN {X 0,Y 219.488,Z 204.764,A -85,B 0,C 180,E1 -21168.071,E2 -21168.071} C_VEL
LIN {X 0,Y 220.53,Z 191.817,A -85,B 0,C 180,E1 -21168.983,E2 -21168.983} C_VEL
LIN {X 0,Y 221.212,Z 177.46,A -85,B 0,C 180,E1 -21169.571,E2 -21169.571} C_VEL
LIN {X 0,Y 223.18,Z 121.298,A -85,B 0,C 180,E1 -21171.316,E2 -21171.316} C_VEL
LIN {X 0,Y 216.722,Z 106.631,A -85,B 0,C 180,E1 -21172.753,E2 -21172.753} C_VEL
LIN {X 0,Y 208.309,Z 90.334,A -85,B 0,C 180,E1 -21174.678,E2 -21174.678} C_VEL
LIN {X 0,Y 207.04,Z 87.969,A -85,B 0,C 180,E1 -21174.981,E2 -21174.981} C_VEL
LIN {X 0,Y 206.779,Z 86.727,A -85,B 0,C 180,E1 -21175.139,E2 -21175.139} C_VEL
LIN {X 0,Y 206.738,Z 86.731,A -85,B 0,C 180,E1 -21178.42,E2 -21178.42} C_VEL
LIN {X 0,Y 206.707,Z 86.737,A -85,B 0,C 180,E1 -21182.957,E2 -21182.957} C_VEL
LIN {X 0,Y 206.723,Z 86.734,A -85,B 0,C 180,E1 -21185.321,E2 -21185.321} C_VEL
LIN {X 0,Y 206.669,Z 86.739,A -85,B 0,C 180,E1 -21190.25,E2 -21190.25} C_VEL
LIN {X 0,Y 206.635,Z 86.742,A -85,B 0,C 180,E1 -21194.419,E2 -21194.419} C_VEL
LIN {X 0,Y 206.662,Z 86.736,A -85,B 0,C 180,E1 -21199.749,E2 -21199.749} C_VEL
LIN {X 0,Y 206.701,Z 86.73,A -85,B 0,C 180,E1 -21204.689,E2 -21204.689} C_VEL
LIN {X 0,Y 206.725,Z 86.728,A -85,B 0,C 180,E1 -21209.34,E2 -21209.34} C_VEL
LIN {X 0,Y 206.736,Z 86.73,A -85,B 0,C 180,E1 -21213.773,E2 -21213.773} C_VEL
LIN {X 0,Y 206.761,Z 86.73,A -85,B 0,C 180,E1 -21218.044,E2 -21218.044} C_VEL
LIN {X 0,Y 206.877,Z 86.694,A -85,B 0,C 180,E1 -21222.197,E2 -21222.197} C_VEL
LIN {X 0,Y 206.899,Z 86.7,A -85,B 0,C 180,E1 -21226.245,E2 -21226.245} C_VEL
LIN {X 0,Y 207.102,Z 86.688,A -85,B 0,C 180,E1 -21230.231,E2 -21230.231} C_VEL
LIN {X 0,Y 207.062,Z 86.669,A -85,B 0,C 180,E1 -21234.156,E2 -21234.156} C_VEL
LIN {X 0,Y 207.384,Z 86.639,A -85,B 0,C 180,E1 -21238.058,E2 -21238.058} C_VEL
LIN {X 0,Y 207.519,Z 86.634,A -85,B 0,C 180,E1 -21240,E2 -21240} C_VEL
LIN {X 0,Y 207.383,Z 86.653,A -85,B 0,C 180,E1 -21241.942,E2 -21241.942} C_VEL
LIN {X 0,Y 207.135,Z 86.683,A -85,B 0,C 180,E1 -21247.8,E2 -21247.8} C_VEL
LIN {X 0,Y 206.921,Z 86.71,A -85,B 0,C 180,E1 -21251.759,E2 -21251.759} C_VEL
LIN {X 0,Y 206.856,Z 86.714,A -85,B 0,C 180,E1 -21255.772,E2 -21255.772} C_VEL
LIN {X 0,Y 206.766,Z 86.725,A -85,B 0,C 180,E1 -21259.871,E2 -21259.871} C_VEL
LIN {X 0,Y 206.743,Z 86.731,A -85,B 0,C 180,E1 -21264.075,E2 -21264.075} C_VEL
LIN {X 0,Y 206.692,Z 86.74,A -85,B 0,C 180,E1 -21268.427,E2 -21268.427} C_VEL
LIN {X 0,Y 206.698,Z 86.741,A -85,B 0,C 180,E1 -21272.958,E2 -21272.958} C_VEL
LIN {X 0,Y 206.683,Z 86.74,A -85,B 0,C 180,E1 -21277.74,E2 -21277.74} C_VEL
LIN {X 0,Y 206.645,Z 86.744,A -85,B 0,C 180,E1 -21281.563,E2 -21281.563} C_VEL
LIN {X 0,Y 206.636,Z 86.745,A -85,B 0,C 180,E1 -21285.582,E2 -21285.582} C_VEL
LIN {X 0,Y 206.725,Z 86.945,A -85,B 0,C 180,E1 -21289.763,E2 -21289.763} C_VEL
LIN {X 0,Y 208.764,Z 95.217,A -85,B 0,C 180,E1 -21293.626,E2 -21293.626} C_VEL
LIN {X 0,Y 209.322,Z 97.7,A -85,B 0,C 180,E1 -21294.412,E2 -21294.412} C_VEL
LIN {X 0,Y 210.126,Z 101.734,A -85,B 0,C 180,E1 -21295.114,E2 -21295.114} C_VEL
LIN {X 0,Y 211.041,Z 108.237,A -85,B 0,C 180,E1 -21295.706,E2 -21295.706} C_VEL
LIN {X 0,Y 212.139,Z 124.831,A -85,B 0,C 180,E1 -21296.508,E2 -21296.508} C_VEL
LIN {X 0,Y 214.48,Z 147.649,A -85,B 0,C 180,E1 -21297.705,E2 -21297.705} C_VEL
LIN {X 0,Y 215.586,Z 160.128,A -85,B 0,C 180,E1 -21298.32,E2 -21298.32} C_VEL
LIN {X 0,Y 213.731,Z 207.728,A -85,B 0,C 180,E1 -21299.879,E2 -21299.879} C_VEL
LIN {X 0,Y 212.583,Z 221.265,A -85,B 0,C 180,E1 -21300.679,E2 -21300.679} C_VEL
LIN {X 0,Y 210.943,Z 233.921,A -85,B 0,C 180,E1 -21301.791,E2 -21301.791} C_VEL
LIN {X 0,Y 208.954,Z 245.964,A -85,B 0,C 180,E1 -21303.265,E2 -21303.265} C_VEL
LIN {X 0,Y 206.55,Z 257.469,A -85,B 0,C 180,E1 -21305.098,E2 -21305.098} C_VEL
LIN {X 0,Y 204.455,Z 267.886,A -85,B 0,C 180,E1 -21307.25,E2 -21307.25} C_VEL
LIN {X 0,Y 202.373,Z 277.209,A -85,B 0,C 180,E1 -21309.679,E2 -21309.679} C_VEL
LIN {X 0,Y 201.413,Z 281.306,A -85,B 0,C 180,E1 -21310.933,E2 -21310.933} C_VEL
LIN {X 0,Y 199.96,Z 288.88,A -85,B 0,C 180,E1 -21313.669,E2 -21313.669} C_VEL
LIN {X 0,Y 198.582,Z 295.625,A -85,B 0,C 180,E1 -21316.7,E2 -21316.7} C_VEL
LIN {X 0,Y 197.844,Z 301.012,A -85,B 0,C 180,E1 -21319.769,E2 -21319.769} C_VEL
LIN {X 0,Y 197.475,Z 305.188,A -85,B 0,C 180,E1 -21322.844,E2 -21322.844} C_VEL
LIN {X 0,Y 197.476,Z 308.28,A -85,B 0,C 180,E1 -21325.918,E2 -21325.918} C_VEL
LIN {X 0,Y 197.605,Z 309.803,A -85,B 0,C 180,E1 -21327.962,E2 -21327.962} C_VEL
LIN {X 0,Y 197.699,Z 310.855,A -85,B 0,C 180,E1 -21330,E2 -21330} C_VEL
LIN {X 0,Y 197.578,Z 311.487,A -85,B 0,C 180,E1 -21332.038,E2 -21332.038} C_VEL
LIN {X 0,Y 197.463,Z 311.724,A -85,B 0,C 180,E1 -21334.749,E2 -21334.749} C_VEL
LIN {X 0,Y 197.514,Z 310.995,A -85,B 0,C 180,E1 -21338.183,E2 -21338.183} C_VEL
LIN {X 0,Y 198.44,Z 308.671,A -85,B 0,C 180,E1 -21342.269,E2 -21342.269} C_VEL
LIN {X 0,Y 199.73,Z 305.847,A -85,B 0,C 180,E1 -21345.302,E2 -21345.302} C_VEL
LIN {X 0,Y 201.693,Z 302.029,A -85,B 0,C 180,E1 -21348.277,E2 -21348.277} C_VEL
LIN {X 0,Y 204.18,Z 297.115,A -85,B 0,C 180,E1 -21351.187,E2 -21351.187} C_VEL
LIN {X 0,Y 206.981,Z 290.956,A -85,B 0,C 180,E1 -21354.045,E2 -21354.045} C_VEL
LIN {X 0,Y 210.559,Z 283.341,A -85,B 0,C 180,E1 -21356.782,E2 -21356.782} C_VEL
LIN {X 0,Y 213.952,Z 275.58,A -85,B 0,C 180,E1 -21358.981,E2 -21358.981} C_VEL
LIN {X 0,Y 218.113,Z 265.064,A -85,B 0,C 180,E1 -21361.304,E2 -21361.304} C_VEL
LIN {X 0,Y 221.365,Z 255.681,A -85,B 0,C 180,E1 -21362.935,E2 -21362.935} C_VEL
LIN {X 0,Y 224.823,Z 244.085,A -85,B 0,C 180,E1 -21364.513,E2 -21364.513} C_VEL
LIN {X 0,Y 227.874,Z 231.761,A -85,B 0,C 180,E1 -21365.737,E2 -21365.737} C_VEL
LIN {X 0,Y 230.321,Z 218.124,A -85,B 0,C 180,E1 -21366.715,E2 -21366.715} C_VEL
LIN {X 0,Y 231.928,Z 204.916,A -85,B 0,C 180,E1 -21367.305,E2 -21367.305} C_VEL
LIN {X 0,Y 233.963,Z 166.02,A -85,B 0,C 180,E1 -21368.474,E2 -21368.474} C_VEL
LIN {X 0,Y 231.881,Z 149.95,A -85,B 0,C 180,E1 -21369.619,E2 -21369.619} C_VEL
LIN {X 0,Y 226.562,Z 137.629,A -85,B 0,C 180,E1 -21371.458,E2 -21371.458} C_VEL
LIN {X 0,Y 221.238,Z 126.642,A -85,B 0,C 180,E1 -21373.391,E2 -21373.391} C_VEL
LIN {X 0,Y 215.624,Z 116.648,A -85,B 0,C 180,E1 -21375.545,E2 -21375.545} C_VEL
LIN {X 0,Y 212.299,Z 111.079,A -85,B 0,C 180,E1 -21376.905,E2 -21376.905} C_VEL
LIN {X 0,Y 209.38,Z 106.341,A -85,B 0,C 180,E1 -21378.163,E2 -21378.163} C_VEL
LIN {X 0,Y 205.704,Z 100.699,A -85,B 0,C 180,E1 -21379.835,E2 -21379.835} C_VEL
LIN {X 0,Y 202.568,Z 96.1,A -85,B 0,C 180,E1 -21381.354,E2 -21381.354} C_VEL
LIN {X 0,Y 202.075,Z 94.93,A -85,B 0,C 180,E1 -21381.72,E2 -21381.72} C_VEL
LIN {X 0,Y 199.67,Z 87.607,A -85,B 0,C 180,E1 -21387.711,E2 -21387.711} C_VEL
LIN {X 0,Y 199.689,Z 87.606,A -85,B 0,C 180,E1 -21392.772,E2 -21392.772} C_VEL
LIN {X 0,Y 199.741,Z 87.596,A -85,B 0,C 180,E1 -21397.229,E2 -21397.229} C_VEL
LIN {X 0,Y 199.84,Z 87.583,A -85,B 0,C 180,E1 -21401.722,E2 -21401.722} C_VEL
LIN {X 0,Y 199.839,Z 87.592,A -85,B 0,C 180,E1 -21405.748,E2 -21405.748} C_VEL
LIN {X 0,Y 200.025,Z 87.567,A -85,B 0,C 180,E1 -21409.882,E2 -21409.882} C_VEL
LIN {X 0,Y 200.025,Z 87.554,A -85,B 0,C 180,E1 -21413.949,E2 -21413.949} C_VEL
LIN {X 0,Y 200.323,Z 87.515,A -85,B 0,C 180,E1 -21417.989,E2 -21417.989} C_VEL
LIN {X 0,Y 200.482,Z 87.505,A -85,B 0,C 180,E1 -21420,E2 -21420} C_VEL
LIN {X 0,Y 200.026,Z 87.552,A -85,B 0,C 180,E1 -21424.029,E2 -21424.029} C_VEL
LIN {X 0,Y 200.088,Z 87.547,A -85,B 0,C 180,E1 -21428.076,E2 -21428.076} C_VEL
LIN {X 0,Y 199.873,Z 87.584,A -85,B 0,C 180,E1 -21432.179,E2 -21432.179} C_VEL
LIN {X 0,Y 199.798,Z 87.598,A -85,B 0,C 180,E1 -21436.344,E2 -21436.344} C_VEL
LIN {X 0,Y 199.683,Z 87.611,A -85,B 0,C 180,E1 -21440.607,E2 -21440.607} C_VEL
LIN {X 0,Y 199.654,Z 87.616,A -85,B 0,C 180,E1 -21444.987,E2 -21444.987} C_VEL
LIN {X 0,Y 199.658,Z 87.623,A -85,B 0,C 180,E1 -21447.642,E2 -21447.642} C_VEL
LIN {X 0,Y 200.511,Z 90.184,A -85,B 0,C 180,E1 -21448.186,E2 -21448.186} C_VEL
LIN {X 0,Y 202.561,Z 92.488,A -85,B 0,C 180,E1 -21449.203,E2 -21449.203} C_VEL
LIN {X 0,Y 203.714,Z 93.378,A -85,B 0,C 180,E1 -21449.731,E2 -21449.731} C_VEL
LIN {X 0,Y 205.665,Z 96.565,A -85,B 0,C 180,E1 -21450.693,E2 -21450.693} C_VEL
LIN {X 0,Y 207.675,Z 98.725,A -85,B 0,C 180,E1 -21451.579,E2 -21451.579} C_VEL
LIN {X 0,Y 210.342,Z 102.351,A -85,B 0,C 180,E1 -21452.742,E2 -21452.742} C_VEL
LIN {X 0,Y 214.894,Z 108.686,A -85,B 0,C 180,E1 -21454.602,E2 -21454.602} C_VEL
LIN {X 0,Y 220.473,Z 116.78,A -85,B 0,C 180,E1 -21456.705,E2 -21456.705} C_VEL
LIN {X 0,Y 227.302,Z 127.796,A -85,B 0,C 180,E1 -21459.08,E2 -21459.08} C_VEL
LIN {X 0,Y 234.365,Z 140.574,A -85,B 0,C 180,E1 -21461.352,E2 -21461.352} C_VEL
LIN {X 0,Y 235.243,Z 142.536,A -85,B 0,C 180,E1 -21461.635,E2 -21461.635} C_VEL
LIN {X 0,Y 232.611,Z 188.304,A -85,B 0,C 180,E1 -21462.992,E2 -21462.992} C_VEL
LIN {X 0,Y 231.17,Z 201.353,A -85,B 0,C 180,E1 -21463.698,E2 -21463.698} C_VEL
LIN {X 0,Y 229.386,Z 212.941,A -85,B 0,C 180,E1 -21464.637,E2 -21464.637} C_VEL
LIN {X 0,Y 226.871,Z 224.582,A -85,B 0,C 180,E1 -21465.875,E2 -21465.875} C_VEL
LIN {X 0,Y 223.702,Z 236.182,A -85,B 0,C 180,E1 -21467.51,E2 -21467.51} C_VEL
LIN {X 0,Y 220.217,Z 246.831,A -85,B 0,C 180,E1 -21469.44,E2 -21469.44} C_VEL
LIN {X 0,Y 216.78,Z 255.999,A -85,B 0,C 180,E1 -21471.56,E2 -21471.56} C_VEL
LIN {X 0,Y 212.966,Z 264.771,A -85,B 0,C 180,E1 -21474.143,E2 -21474.143} C_VEL
LIN {X 0,Y 209.417,Z 272.352,A -85,B 0,C 180,E1 -21477.034,E2 -21477.034} C_VEL
LIN {X 0,Y 205.933,Z 278.92,A -85,B 0,C 180,E1 -21480.34,E2 -21480.34} C_VEL
LIN {X 0,Y 203.415,Z 283.314,A -85,B 0,C 180,E1 -21483.311,E2 -21483.311} C_VEL
LIN {X 0,Y 202.023,Z 285.617,A -85,B 0,C 180,E1 -21485.326,E2 -21485.326} C_VEL
LIN {X 0,Y 200.807,Z 287.476,A -85,B 0,C 180,E1 -21487.357,E2 -21487.357} C_VEL
LIN {X 0,Y 199.805,Z 288.85,A -85,B 0,C 180,E1 -21489.406,E2 -21489.406} C_VEL
LIN {X 0,Y 198.412,Z 290.374,A -85,B 0,C 180,E1 -21493.539,E2 -21493.539} C_VEL
LIN {X 0,Y 197.931,Z 290.534,A -85,B 0,C 180,E1 -21495.608,E2 -21495.608} C_VEL
LIN {X 0,Y 197.475,Z 289.596,A -85,B 0,C 180,E1 -21499.75,E2 -21499.75} C_VEL
LIN {X 0,Y 197.513,Z 288.543,A -85,B 0,C 180,E1 -21501.817,E2 -21501.817} C_VEL
LIN {X 0,Y 197.829,Z 286.857,A -85,B 0,C 180,E1 -21504.107,E2 -21504.107} C_VEL
LIN {X 0,Y 198.133,Z 284.051,A -85,B 0,C 180,E1 -21506.95,E2 -21506.95} C_VEL
LIN {X 0,Y 198.844,Z 280.001,A -85,B 0,C 180,E1 -21510,E2 -21510} C_VEL
LIN {X 0,Y 199.974,Z 273.804,A -85,B 0,C 180,E1 -21513.526,E2 -21513.526} C_VEL
LIN {X 0,Y 201.594,Z 267.041,A -85,B 0,C 180,E1 -21516.506,E2 -21516.506} C_VEL
LIN {X 0,Y 203.459,Z 258.656,A -85,B 0,C 180,E1 -21519.444,E2 -21519.444} C_VEL
LIN {X 0,Y 205.396,Z 250.013,A -85,B 0,C 180,E1 -21521.847,E2 -21521.847} C_VEL
LIN {X 0,Y 207.619,Z 240.5,A -85,B 0,C 180,E1 -21523.957,E2 -21523.957} C_VEL
LIN {X 0,Y 209.614,Z 230.156,A -85,B 0,C 180,E1 -21525.808,E2 -21525.808} C_VEL
LIN {X 0,Y 211.423,Z 218.835,A -85,B 0,C 180,E1 -21527.408,E2 -21527.408} C_VEL
LIN {X 0,Y 212.827,Z 207.224,A -85,B 0,C 180,E1 -21528.657,E2 -21528.657} C_VEL
LIN {X 0,Y 214.018,Z 193.78,A -85,B 0,C 180,E1 -21529.676,E2 -21529.676} C_VEL
LIN {X 0,Y 214.725,Z 180.844,A -85,B 0,C 180,E1 -21530.282,E2 -21530.282} C_VEL
LIN {X 0,Y 216.886,Z 123.185,A -85,B 0,C 180,E1 -21532.114,E2 -21532.114} C_VEL
LIN {X 0,Y 210.245,Z 108.292,A -85,B 0,C 180,E1 -21533.667,E2 -21533.667} C_VEL
LIN {X 0,Y 202.782,Z 94.002,A -85,B 0,C 180,E1 -21535.461,E2 -21535.461} C_VEL
LIN {X 0,Y 199.971,Z 88.898,A -85,B 0,C 180,E1 -21536.169,E2 -21536.169} C_VEL
LIN {X 0,Y 199.706,Z 87.609,A -85,B 0,C 180,E1 -21536.345,E2 -21536.345} C_VEL
LIN {X 0,Y 199.666,Z 87.614,A -85,B 0,C 180,E1 -21539.524,E2 -21539.524} C_VEL
LIN {X 0,Y 199.66,Z 87.616,A -85,B 0,C 180,E1 -21542.35,E2 -21542.35} C_VEL
LIN {X 0,Y 199.641,Z 87.615,A -85,B 0,C 180,E1 -21546.76,E2 -21546.76} C_VEL
LIN {X 0,Y 199.64,Z 87.617,A -85,B 0,C 180,E1 -21549.321,E2 -21549.321} C_VEL
LIN {X 0,Y 199.581,Z 87.62,A -85,B 0,C 180,E1 -21554.772,E2 -21554.772} C_VEL
LIN {X 0,Y 199.58,Z 87.621,A -85,B 0,C 180,E1 -21558.005,E2 -21558.005} C_VEL
LIN {X 0,Y 199.612,Z 87.615,A -85,B 0,C 180,E1 -21560.768,E2 -21560.768} C_VEL
LIN {X 0,Y 199.616,Z 87.617,A -85,B 0,C 180,E1 -21565.714,E2 -21565.714} C_VEL
LIN {X 0,Y 199.703,Z 87.606,A -85,B 0,C 180,E1 -21568.138,E2 -21568.138} C_VEL
LIN {X 0,Y 199.69,Z 87.612,A -85,B 0,C 180,E1 -21572.772,E2 -21572.772} C_VEL
LIN {X 0,Y 199.741,Z 87.604,A -85,B 0,C 180,E1 -21577.23,E2 -21577.23} C_VEL
LIN {X 0,Y 199.8,Z 87.579,A -85,B 0,C 180,E1 -21581.758,E2 -21581.758} C_VEL
LIN {X 0,Y 199.839,Z 87.577,A -85,B 0,C 180,E1 -21585.749,E2 -21585.749} C_VEL
LIN {X 0,Y 200.025,Z 87.57,A -85,B 0,C 180,E1 -21589.882,E2 -21589.882} C_VEL
LIN {X 0,Y 200.024,Z 87.546,A -85,B 0,C 180,E1 -21593.95,E2 -21593.95} C_VEL
LIN {X 0,Y 200.323,Z 87.517,A -85,B 0,C 180,E1 -21597.99,E2 -21597.99} C_VEL
LIN {X 0,Y 200.483,Z 87.51,A -85,B 0,C 180,E1 -21600,E2 -21600} C_VEL
LIN {X 0,Y 200.023,Z 87.562,A -85,B 0,C 180,E1 -21604.03,E2 -21604.03} C_VEL
LIN {X 0,Y 200.085,Z 87.56,A -85,B 0,C 180,E1 -21608.077,E2 -21608.077} C_VEL
LIN {X 0,Y 199.871,Z 87.587,A -85,B 0,C 180,E1 -21612.18,E2 -21612.18} C_VEL
LIN {X 0,Y 199.797,Z 87.594,A -85,B 0,C 180,E1 -21616.344,E2 -21616.344} C_VEL
LIN {X 0,Y 199.684,Z 87.607,A -85,B 0,C 180,E1 -21620.607,E2 -21620.607} C_VEL
LIN {X 0,Y 199.655,Z 87.613,A -85,B 0,C 180,E1 -21624.987,E2 -21624.987} C_VEL
LIN {X 0,Y 199.612,Z 87.622,A -85,B 0,C 180,E1 -21629.533,E2 -21629.533} C_VEL
LIN {X 0,Y 199.668,Z 87.616,A -85,B 0,C 180,E1 -21632.353,E2 -21632.353} C_VEL
LIN {X 0,Y 199.626,Z 87.621,A -85,B 0,C 180,E1 -21636.763,E2 -21636.763} C_VEL
LIN {X 0,Y 199.611,Z 87.62,A -85,B 0,C 180,E1 -21639.328,E2 -21639.328} C_VEL
LIN {X 0,Y 199.577,Z 87.624,A -85,B 0,C 180,E1 -21642.31,E2 -21642.31} C_VEL
LIN {X 0,Y 199.582,Z 87.624,A -85,B 0,C 180,E1 -21645.229,E2 -21645.229} C_VEL
LIN {X 0,Y 199.643,Z 87.665,A -85,B 0,C 180,E1 -21648.815,E2 -21648.815} C_VEL
LIN {X 0,Y 201.518,Z 95.22,A -85,B 0,C 180,E1 -21652.52,E2 -21652.52} C_VEL
LIN {X 0,Y 202.19,Z 98.067,A -85,B 0,C 180,E1 -21653.852,E2 -21653.852} C_VEL
LIN {X 0,Y 209.176,Z 114.97,A -85,B 0,C 180,E1 -21655.677,E2 -21655.677} C_VEL
LIN {X 0,Y 211.914,Z 122.402,A -85,B 0,C 180,E1 -21656.382,E2 -21656.382} C_VEL
LIN {X 0,Y 212.139,Z 124.831,A -85,B 0,C 180,E1 -21656.508,E2 -21656.508} C_VEL
LIN {X 0,Y 212.28,Z 130.662,A -85,B 0,C 180,E1 -21656.75,E2 -21656.75} C_VEL
LIN {X 0,Y 210.741,Z 140.449,A -85,B 0,C 180,E1 -21656.896,E2 -21656.896} C_VEL
LIN {X 0,Y 209.051,Z 150.264,A -85,B 0,C 180,E1 -21657.023,E2 -21657.023} C_VEL
LIN {X 0,Y 208.971,Z 156.149,A -85,B 0,C 180,E1 -21657.237,E2 -21657.237} C_VEL
LIN {X 0,Y 209.21,Z 161.758,A -85,B 0,C 180,E1 -21657.487,E2 -21657.487} C_VEL
LIN {X 0,Y 207.374,Z 207.331,A -85,B 0,C 180,E1 -21659.022,E2 -21659.022} C_VEL
LIN {X 0,Y 206.197,Z 220.58,A -85,B 0,C 180,E1 -21659.818,E2 -21659.818} C_VEL
LIN {X 0,Y 204.516,Z 233.325,A -85,B 0,C 180,E1 -21660.961,E2 -21660.961} C_VEL
LIN {X 0,Y 202.555,Z 244.62,A -85,B 0,C 180,E1 -21662.35,E2 -21662.35} C_VEL
LIN {X 0,Y 200.133,Z 256.315,A -85,B 0,C 180,E1 -21664.242,E2 -21664.242} C_VEL
LIN {X 0,Y 197.813,Z 266.854,A -85,B 0,C 180,E1 -21666.441,E2 -21666.441} C_VEL
LIN {X 0,Y 195.704,Z 276.337,A -85,B 0,C 180,E1 -21668.954,E2 -21668.954} C_VEL
LIN {X 0,Y 194.451,Z 281.329,A -85,B 0,C 180,E1 -21670.535,E2 -21670.535} C_VEL
LIN {X 0,Y 192.832,Z 289.374,A -85,B 0,C 180,E1 -21673.593,E2 -21673.593} C_VEL
LIN {X 0,Y 191.639,Z 294.937,A -85,B 0,C 180,E1 -21676.209,E2 -21676.209} C_VEL
LIN {X 0,Y 190.81,Z 300.383,A -85,B 0,C 180,E1 -21679.387,E2 -21679.387} C_VEL
LIN {X 0,Y 190.42,Z 304.618,A -85,B 0,C 180,E1 -21682.578,E2 -21682.578} C_VEL
LIN {X 0,Y 190.405,Z 307.763,A -85,B 0,C 180,E1 -21685.766,E2 -21685.766} C_VEL
LIN {X 0,Y 190.513,Z 309.319,A -85,B 0,C 180,E1 -21687.886,E2 -21687.886} C_VEL
LIN {X 0,Y 190.631,Z 310.412,A -85,B 0,C 180,E1 -21690,E2 -21690} C_VEL
LIN {X 0,Y 190.488,Z 311.066,A -85,B 0,C 180,E1 -21692.114,E2 -21692.114} C_VEL
LIN {X 0,Y 190.4,Z 311.352,A -85,B 0,C 180,E1 -21694.71,E2 -21694.71} C_VEL
LIN {X 0,Y 190.469,Z 310.668,A -85,B 0,C 180,E1 -21698.487,E2 -21698.487} C_VEL
LIN {X 0,Y 191.467,Z 308.391,A -85,B 0,C 180,E1 -21702.723,E2 -21702.723} C_VEL
LIN {X 0,Y 192.869,Z 305.619,A -85,B 0,C 180,E1 -21705.86,E2 -21705.86} C_VEL
LIN {X 0,Y 194.924,Z 301.854,A -85,B 0,C 180,E1 -21708.935,E2 -21708.935} C_VEL
LIN {X 0,Y 197.543,Z 296.997,A -85,B 0,C 180,E1 -21711.935,E2 -21711.935} C_VEL
LIN {X 0,Y 201.091,Z 289.778,A -85,B 0,C 180,E1 -21715.349,E2 -21715.349} C_VEL
LIN {X 0,Y 204.928,Z 281.928,A -85,B 0,C 180,E1 -21718.135,E2 -21718.135} C_VEL
LIN {X 0,Y 209.313,Z 272.169,A -85,B 0,C 180,E1 -21720.8,E2 -21720.8} C_VEL
LIN {X 0,Y 213.348,Z 262.083,A -85,B 0,C 180,E1 -21722.925,E2 -21722.925} C_VEL
LIN {X 0,Y 216.389,Z 253.488,A -85,B 0,C 180,E1 -21724.355,E2 -21724.355} C_VEL
LIN {X 0,Y 219.526,Z 243.043,A -85,B 0,C 180,E1 -21725.751,E2 -21725.751} C_VEL
LIN {X 0,Y 222.668,Z 230.487,A -85,B 0,C 180,E1 -21726.989,E2 -21726.989} C_VEL
LIN {X 0,Y 225.07,Z 217.27,A -85,B 0,C 180,E1 -21727.935,E2 -21727.935} C_VEL
LIN {X 0,Y 226.649,Z 204.754,A -85,B 0,C 180,E1 -21728.49,E2 -21728.49} C_VEL
LIN {X 0,Y 228.73,Z 167.059,A -85,B 0,C 180,E1 -21729.639,E2 -21729.639} C_VEL
LIN {X 0,Y 226.913,Z 152.814,A -85,B 0,C 180,E1 -21730.699,E2 -21730.699} C_VEL
LIN {X 0,Y 221.087,Z 139.28,A -85,B 0,C 180,E1 -21732.84,E2 -21732.84} C_VEL
LIN {X 0,Y 215.292,Z 127.582,A -85,B 0,C 180,E1 -21735.097,E2 -21735.097} C_VEL
LIN {X 0,Y 208.892,Z 116.426,A -85,B 0,C 180,E1 -21737.779,E2 -21737.779} C_VEL
LIN {X 0,Y 205.964,Z 111.597,A -85,B 0,C 180,E1 -21739.105,E2 -21739.105} C_VEL
LIN {X 0,Y 202.594,Z 106.299,A -85,B 0,C 180,E1 -21740.721,E2 -21740.721} C_VEL
LIN {X 0,Y 199.357,Z 101.293,A -85,B 0,C 180,E1 -21742.387,E2 -21742.387} C_VEL
LIN {X 0,Y 195.227,Z 95.717,A -85,B 0,C 180,E1 -21744.662,E2 -21744.662} C_VEL
LIN {X 0,Y 194.489,Z 94.296,A -85,B 0,C 180,E1 -21745.153,E2 -21745.153} C_VEL
LIN {X 0,Y 193.386,Z 90.86,A -85,B 0,C 180,E1 -21748.2,E2 -21748.2} C_VEL
LIN {X 0,Y 192.654,Z 88.477,A -85,B 0,C 180,E1 -21750.556,E2 -21750.556} C_VEL
LIN {X 0,Y 192.709,Z 88.481,A -85,B 0,C 180,E1 -21756.349,E2 -21756.349} C_VEL
LIN {X 0,Y 192.784,Z 88.464,A -85,B 0,C 180,E1 -21761.414,E2 -21761.414} C_VEL
LIN {X 0,Y 192.767,Z 88.474,A -85,B 0,C 180,E1 -21765.214,E2 -21765.214} C_VEL
LIN {X 0,Y 192.947,Z 88.444,A -85,B 0,C 180,E1 -21769.566,E2 -21769.566} C_VEL
LIN {X 0,Y 192.987,Z 88.429,A -85,B 0,C 180,E1 -21773.728,E2 -21773.728} C_VEL
LIN {X 0,Y 193.265,Z 88.394,A -85,B 0,C 180,E1 -21777.916,E2 -21777.916} C_VEL
LIN {X 0,Y 193.446,Z 88.38,A -85,B 0,C 180,E1 -21780,E2 -21780} C_VEL
LIN {X 0,Y 192.972,Z 88.431,A -85,B 0,C 180,E1 -21784.177,E2 -21784.177} C_VEL
LIN {X 0,Y 193.036,Z 88.424,A -85,B 0,C 180,E1 -21788.374,E2 -21788.374} C_VEL
LIN {X 0,Y 192.8,Z 88.46,A -85,B 0,C 180,E1 -21792.633,E2 -21792.633} C_VEL
LIN {X 0,Y 192.754,Z 88.472,A -85,B 0,C 180,E1 -21796.959,E2 -21796.959} C_VEL
LIN {X 0,Y 192.616,Z 88.49,A -85,B 0,C 180,E1 -21801.399,E2 -21801.399} C_VEL
LIN {X 0,Y 192.67,Z 88.65,A -85,B 0,C 180,E1 -21804.313,E2 -21804.313} C_VEL
LIN {X 0,Y 193.396,Z 90.963,A -85,B 0,C 180,E1 -21804.864,E2 -21804.864} C_VEL
LIN {X 0,Y 195.293,Z 93.245,A -85,B 0,C 180,E1 -21805.982,E2 -21805.982} C_VEL
LIN {X 0,Y 196.935,Z 94.352,A -85,B 0,C 180,E1 -21806.845,E2 -21806.845} C_VEL
LIN {X 0,Y 198.836,Z 97.554,A -85,B 0,C 180,E1 -21807.926,E2 -21807.926} C_VEL
LIN {X 0,Y 201.055,Z 99.782,A -85,B 0,C 180,E1 -21809.028,E2 -21809.028} C_VEL
LIN {X 0,Y 203.656,Z 103.387,A -85,B 0,C 180,E1 -21810.311,E2 -21810.311} C_VEL
LIN {X 0,Y 205.014,Z 105.132,A -85,B 0,C 180,E1 -21810.944,E2 -21810.944} C_VEL
LIN {X 0,Y 209.648,Z 111.463,A -85,B 0,C 180,E1 -21812.998,E2 -21812.998} C_VEL
LIN {X 0,Y 216.254,Z 121.093,A -85,B 0,C 180,E1 -21815.658,E2 -21815.658} C_VEL
LIN {X 0,Y 222.995,Z 132.115,A -85,B 0,C 180,E1 -21818.135,E2 -21818.135} C_VEL
LIN {X 0,Y 229.958,Z 144.891,A -85,B 0,C 180,E1 -21820.491,E2 -21820.491} C_VEL
LIN {X 0,Y 227.337,Z 188.722,A -85,B 0,C 180,E1 -21821.813,E2 -21821.813} C_VEL
LIN {X 0,Y 225.866,Z 201.598,A -85,B 0,C 180,E1 -21822.519,E2 -21822.519} C_VEL
LIN {X 0,Y 223.766,Z 214.48,A -85,B 0,C 180,E1 -21823.586,E2 -21823.586} C_VEL
LIN {X 0,Y 221.156,Z 225.756,A -85,B 0,C 180,E1 -21824.835,E2 -21824.835} C_VEL
LIN {X 0,Y 217.977,Z 236.836,A -85,B 0,C 180,E1 -21826.435,E2 -21826.435} C_VEL
LIN {X 0,Y 214.346,Z 247.435,A -85,B 0,C 180,E1 -21828.397,E2 -21828.397} C_VEL
LIN {X 0,Y 210.619,Z 256.889,A -85,B 0,C 180,E1 -21830.654,E2 -21830.654} C_VEL
LIN {X 0,Y 206.453,Z 265.976,A -85,B 0,C 180,E1 -21833.435,E2 -21833.435} C_VEL
LIN {X 0,Y 202.849,Z 273.244,A -85,B 0,C 180,E1 -21836.334,E2 -21836.334} C_VEL
LIN {X 0,Y 199.626,Z 278.979,A -85,B 0,C 180,E1 -21839.304,E2 -21839.304} C_VEL
LIN {X 0,Y 196.929,Z 283.45,A -85,B 0,C 180,E1 -21842.358,E2 -21842.358} C_VEL
LIN {X 0,Y 195.421,Z 285.79,A -85,B 0,C 180,E1 -21844.433,E2 -21844.433} C_VEL
LIN {X 0,Y 194.116,Z 287.688,A -85,B 0,C 180,E1 -21846.531,E2 -21846.531} C_VEL
LIN {X 0,Y 193.011,Z 289.127,A -85,B 0,C 180,E1 -21848.646,E2 -21848.646} C_VEL
LIN {X 0,Y 191.482,Z 290.716,A -85,B 0,C 180,E1 -21852.925,E2 -21852.925} C_VEL
LIN {X 0,Y 190.944,Z 290.925,A -85,B 0,C 180,E1 -21855.07,E2 -21855.07} C_VEL
LIN {X 0,Y 190.538,Z 290.7,A -85,B 0,C 180,E1 -21857.214,E2 -21857.214} C_VEL
LIN {X 0,Y 190.418,Z 289.045,A -85,B 0,C 180,E1 -21861.51,E2 -21861.51} C_VEL
LIN {X 0,Y 190.736,Z 287.168,A -85,B 0,C 180,E1 -21864.188,E2 -21864.188} C_VEL
LIN {X 0,Y 191.169,Z 283.444,A -85,B 0,C 180,E1 -21867.893,E2 -21867.893} C_VEL
LIN {X 0,Y 192.028,Z 279.099,A -85,B 0,C 180,E1 -21871.049,E2 -21871.049} C_VEL
LIN {X 0,Y 193.131,Z 273.587,A -85,B 0,C 180,E1 -21874.174,E2 -21874.174} C_VEL
LIN {X 0,Y 194.87,Z 266.689,A -85,B 0,C 180,E1 -21877.252,E2 -21877.252} C_VEL
LIN {X 0,Y 196.88,Z 258.07,A -85,B 0,C 180,E1 -21880.282,E2 -21880.282} C_VEL
LIN {X 0,Y 198.944,Z 249.233,A -85,B 0,C 180,E1 -21882.756,E2 -21882.756} C_VEL
LIN {X 0,Y 201.288,Z 239.484,A -85,B 0,C 180,E1 -21884.922,E2 -21884.922} C_VEL
LIN {X 0,Y 203.397,Z 228.822,A -85,B 0,C 180,E1 -21886.821,E2 -21886.821} C_VEL
LIN {X 0,Y 205.263,Z 216.908,A -85,B 0,C 180,E1 -21888.464,E2 -21888.464} C_VEL
LIN {X 0,Y 206.737,Z 204.534,A -85,B 0,C 180,E1 -21889.745,E2 -21889.745} C_VEL
LIN {X 0,Y 207.796,Z 192.097,A -85,B 0,C 180,E1 -21890.645,E2 -21890.645} C_VEL
LIN {X 0,Y 208.534,Z 177.491,A -85,B 0,C 180,E1 -21891.259,E2 -21891.259} C_VEL
LIN {X 0,Y 210.542,Z 124.853,A -85,B 0,C 180,E1 -21892.982,E2 -21892.982} C_VEL
LIN {X 0,Y 203.644,Z 109.591,A -85,B 0,C 180,E1 -21894.68,E2 -21894.68} C_VEL
LIN {X 0,Y 196.072,Z 95.363,A -85,B 0,C 180,E1 -21896.613,E2 -21896.613} C_VEL
LIN {X 0,Y 193.911,Z 91.741,A -85,B 0,C 180,E1 -21897.181,E2 -21897.181} C_VEL
LIN {X 0,Y 192.724,Z 89.009,A -85,B 0,C 180,E1 -21897.533,E2 -21897.533} C_VEL
LIN {X 0,Y 192.659,Z 88.486,A -85,B 0,C 180,E1 -21897.664,E2 -21897.664} C_VEL
LIN {X 0,Y 192.599,Z 88.495,A -85,B 0,C 180,E1 -21903.186,E2 -21903.186} C_VEL
LIN {X 0,Y 192.611,Z 88.491,A -85,B 0,C 180,E1 -21906.608,E2 -21906.608} C_VEL
LIN {X 0,Y 192.525,Z 88.498,A -85,B 0,C 180,E1 -21911.078,E2 -21911.078} C_VEL
LIN {X 0,Y 192.492,Z 88.503,A -85,B 0,C 180,E1 -21916.076,E2 -21916.076} C_VEL
LIN {X 0,Y 192.519,Z 88.497,A -85,B 0,C 180,E1 -21920.052,E2 -21920.052} C_VEL
LIN {X 0,Y 192.562,Z 88.491,A -85,B 0,C 180,E1 -21924.271,E2 -21924.271} C_VEL
LIN {X 0,Y 192.612,Z 88.493,A -85,B 0,C 180,E1 -21927.059,E2 -21927.059} C_VEL
LIN {X 0,Y 192.667,Z 88.484,A -85,B 0,C 180,E1 -21931.693,E2 -21931.693} C_VEL
LIN {X 0,Y 192.709,Z 88.476,A -85,B 0,C 180,E1 -21936.349,E2 -21936.349} C_VEL
LIN {X 0,Y 192.735,Z 88.461,A -85,B 0,C 180,E1 -21941.458,E2 -21941.458} C_VEL
LIN {X 0,Y 192.767,Z 88.45,A -85,B 0,C 180,E1 -21945.214,E2 -21945.214} C_VEL
LIN {X 0,Y 192.948,Z 88.45,A -85,B 0,C 180,E1 -21949.567,E2 -21949.567} C_VEL
LIN {X 0,Y 192.986,Z 88.423,A -85,B 0,C 180,E1 -21953.728,E2 -21953.728} C_VEL
LIN {X 0,Y 193.264,Z 88.395,A -85,B 0,C 180,E1 -21957.916,E2 -21957.916} C_VEL
LIN {X 0,Y 193.447,Z 88.386,A -85,B 0,C 180,E1 -21960,E2 -21960} C_VEL
LIN {X 0,Y 192.968,Z 88.441,A -85,B 0,C 180,E1 -21964.177,E2 -21964.177} C_VEL
LIN {X 0,Y 193.034,Z 88.438,A -85,B 0,C 180,E1 -21968.374,E2 -21968.374} C_VEL
LIN {X 0,Y 192.799,Z 88.468,A -85,B 0,C 180,E1 -21972.634,E2 -21972.634} C_VEL
LIN {X 0,Y 192.754,Z 88.473,A -85,B 0,C 180,E1 -21976.959,E2 -21976.959} C_VEL
LIN {X 0,Y 192.618,Z 88.491,A -85,B 0,C 180,E1 -21981.4,E2 -21981.4} C_VEL
LIN {X 0,Y 192.644,Z 88.488,A -85,B 0,C 180,E1 -21984.209,E2 -21984.209} C_VEL
LIN {X 0,Y 192.605,Z 88.497,A -85,B 0,C 180,E1 -21988.866,E2 -21988.866} C_VEL
LIN {X 0,Y 192.597,Z 88.497,A -85,B 0,C 180,E1 -21993.186,E2 -21993.186} C_VEL
LIN {X 0,Y 192.554,Z 88.501,A -85,B 0,C 180,E1 -21998.352,E2 -21998.352} C_VEL
LIN {X 0,Y 192.494,Z 88.504,A -85,B 0,C 180,E1 -22003.096,E2 -22003.096} C_VEL
LIN {X 0,Y 192.547,Z 88.509,A -85,B 0,C 180,E1 -22007.85,E2 -22007.85} C_VEL
LIN {X 0,Y 194.677,Z 96.865,A -85,B 0,C 180,E1 -22012.141,E2 -22012.141} C_VEL
LIN {X 0,Y 194.861,Z 97.698,A -85,B 0,C 180,E1 -22012.511,E2 -22012.511} C_VEL
LIN {X 0,Y 200.738,Z 111.221,A -85,B 0,C 180,E1 -22014.141,E2 -22014.141} C_VEL
LIN {X 0,Y 205.746,Z 124.159,A -85,B 0,C 180,E1 -22015.496,E2 -22015.496} C_VEL
LIN {X 0,Y 208.218,Z 148.247,A -85,B 0,C 180,E1 -22016.821,E2 -22016.821} C_VEL
LIN {X 0,Y 208.971,Z 156.149,A -85,B 0,C 180,E1 -22017.237,E2 -22017.237} C_VEL
LIN {X 0,Y 208.932,Z 160.029,A -85,B 0,C 180,E1 -22017.38,E2 -22017.38} C_VEL
LIN {X 0,Y 208.285,Z 163.901,A -85,B 0,C 180,E1 -22017.434,E2 -22017.434} C_VEL
LIN {X 0,Y 202.834,Z 181.06,A -85,B 0,C 180,E1 -22017.295,E2 -22017.295} C_VEL
LIN {X 0,Y 201.967,Z 186.96,A -85,B 0,C 180,E1 -22017.398,E2 -22017.398} C_VEL
LIN {X 0,Y 200.949,Z 208.461,A -85,B 0,C 180,E1 -22018.19,E2 -22018.19} C_VEL
LIN {X 0,Y 199.711,Z 221.441,A -85,B 0,C 180,E1 -22019.024,E2 -22019.024} C_VEL
LIN {X 0,Y 197.954,Z 233.805,A -85,B 0,C 180,E1 -22020.195,E2 -22020.195} C_VEL
LIN {X 0,Y 195.938,Z 244.883,A -85,B 0,C 180,E1 -22021.623,E2 -22021.623} C_VEL
LIN {X 0,Y 193.429,Z 256.459,A -85,B 0,C 180,E1 -22023.571,E2 -22023.571} C_VEL
LIN {X 0,Y 191.03,Z 266.907,A -85,B 0,C 180,E1 -22025.839,E2 -22025.839} C_VEL
LIN {X 0,Y 189.053,Z 275.452,A -85,B 0,C 180,E1 -22028.176,E2 -22028.176} C_VEL
LIN {X 0,Y 187.67,Z 280.011,A -85,B 0,C 180,E1 -22029.626,E2 -22029.626} C_VEL
LIN {X 0,Y 186.85,Z 284.694,A -85,B 0,C 180,E1 -22031.354,E2 -22031.354} C_VEL
LIN {X 0,Y 185.2,Z 292.131,A -85,B 0,C 180,E1 -22034.595,E2 -22034.595} C_VEL
LIN {X 0,Y 184.024,Z 298.081,A -85,B 0,C 180,E1 -22037.875,E2 -22037.875} C_VEL
LIN {X 0,Y 183.465,Z 302.767,A -85,B 0,C 180,E1 -22041.186,E2 -22041.186} C_VEL
LIN {X 0,Y 183.331,Z 307.044,A -85,B 0,C 180,E1 -22045.355,E2 -22045.355} C_VEL
LIN {X 0,Y 183.425,Z 308.826,A -85,B 0,C 180,E1 -22047.804,E2 -22047.804} C_VEL
LIN {X 0,Y 183.563,Z 309.969,A -85,B 0,C 180,E1 -22050,E2 -22050} C_VEL
LIN {X 0,Y 183.401,Z 310.646,A -85,B 0,C 180,E1 -22052.196,E2 -22052.196} C_VEL
LIN {X 0,Y 183.325,Z 310.942,A -85,B 0,C 180,E1 -22054.62,E2 -22054.62} C_VEL
LIN {X 0,Y 183.415,Z 310.334,A -85,B 0,C 180,E1 -22058.816,E2 -22058.816} C_VEL
LIN {X 0,Y 184.494,Z 308.111,A -85,B 0,C 180,E1 -22063.212,E2 -22063.212} C_VEL
LIN {X 0,Y 186.034,Z 305.39,A -85,B 0,C 180,E1 -22066.459,E2 -22066.459} C_VEL
LIN {X 0,Y 188.192,Z 301.678,A -85,B 0,C 180,E1 -22069.64,E2 -22069.64} C_VEL
LIN {X 0,Y 191.221,Z 296.301,A -85,B 0,C 180,E1 -22073.062,E2 -22073.062} C_VEL
LIN {X 0,Y 194.69,Z 289.729,A -85,B 0,C 180,E1 -22076.245,E2 -22076.245} C_VEL
LIN {X 0,Y 198.705,Z 281.992,A -85,B 0,C 180,E1 -22079.099,E2 -22079.099} C_VEL
LIN {X 0,Y 202.445,Z 274.108,A -85,B 0,C 180,E1 -22081.382,E2 -22081.382} C_VEL
LIN {X 0,Y 206.965,Z 263.447,A -85,B 0,C 180,E1 -22083.783,E2 -22083.783} C_VEL
LIN {X 0,Y 210.094,Z 255.18,A -85,B 0,C 180,E1 -22085.243,E2 -22085.243} C_VEL
LIN {X 0,Y 213.834,Z 243.646,A -85,B 0,C 180,E1 -22086.857,E2 -22086.857} C_VEL
LIN {X 0,Y 217.068,Z 231.475,A -85,B 0,C 180,E1 -22088.111,E2 -22088.111} C_VEL
LIN {X 0,Y 219.679,Z 217.977,A -85,B 0,C 180,E1 -22089.113,E2 -22089.113} C_VEL
LIN {X 0,Y 221.406,Z 205.36,A -85,B 0,C 180,E1 -22089.706,E2 -22089.706} C_VEL
LIN {X 0,Y 223.598,Z 168.079,A -85,B 0,C 180,E1 -22090.859,E2 -22090.859} C_VEL
LIN {X 0,Y 222.088,Z 155.898,A -85,B 0,C 180,E1 -22091.801,E2 -22091.801} C_VEL
LIN {X 0,Y 215.846,Z 141.271,A -85,B 0,C 180,E1 -22094.248,E2 -22094.248} C_VEL
LIN {X 0,Y 210.631,Z 130.945,A -85,B 0,C 180,E1 -22096.408,E2 -22096.408} C_VEL
LIN {X 0,Y 205.538,Z 121.758,A -85,B 0,C 180,E1 -22098.681,E2 -22098.681} C_VEL
LIN {X 0,Y 202.275,Z 116.327,A -85,B 0,C 180,E1 -22100.243,E2 -22100.243} C_VEL
LIN {X 0,Y 199.331,Z 111.613,A -85,B 0,C 180,E1 -22101.74,E2 -22101.74} C_VEL
LIN {X 0,Y 195.781,Z 106.103,A -85,B 0,C 180,E1 -22103.679,E2 -22103.679} C_VEL
LIN {X 0,Y 192.24,Z 100.93,A -85,B 0,C 180,E1 -22105.784,E2 -22105.784} C_VEL
LIN {X 0,Y 187.444,Z 94.512,A -85,B 0,C 180,E1 -22108.967,E2 -22108.967} C_VEL
LIN {X 0,Y 186.821,Z 93.389,A -85,B 0,C 180,E1 -22109.48,E2 -22109.48} C_VEL
LIN {X 0,Y 186.579,Z 92.129,A -85,B 0,C 180,E1 -22110.68,E2 -22110.68} C_VEL
LIN {X 0,Y 185.565,Z 89.358,A -85,B 0,C 180,E1 -22113.879,E2 -22113.879} C_VEL
LIN {X 0,Y 185.602,Z 89.353,A -85,B 0,C 180,E1 -22117.749,E2 -22117.749} C_VEL
LIN {X 0,Y 185.719,Z 89.336,A -85,B 0,C 180,E1 -22122.378,E2 -22122.378} C_VEL
LIN {X 0,Y 185.732,Z 89.336,A -85,B 0,C 180,E1 -22126.877,E2 -22126.877} C_VEL
LIN {X 0,Y 185.986,Z 89.311,A -85,B 0,C 180,E1 -22131.306,E2 -22131.306} C_VEL
LIN {X 0,Y 186.209,Z 89.273,A -85,B 0,C 180,E1 -22137.837,E2 -22137.837} C_VEL
LIN {X 0,Y 186.409,Z 89.256,A -85,B 0,C 180,E1 -22140,E2 -22140} C_VEL
LIN {X 0,Y 185.918,Z 89.31,A -85,B 0,C 180,E1 -22144.336,E2 -22144.336} C_VEL
LIN {X 0,Y 185.983,Z 89.301,A -85,B 0,C 180,E1 -22148.694,E2 -22148.694} C_VEL
LIN {X 0,Y 185.727,Z 89.337,A -85,B 0,C 180,E1 -22153.123,E2 -22153.123} C_VEL
LIN {X 0,Y 185.688,Z 89.345,A -85,B 0,C 180,E1 -22157.625,E2 -22157.625} C_VEL
LIN {X 0,Y 185.594,Z 89.513,A -85,B 0,C 180,E1 -22160.215,E2 -22160.215} C_VEL
LIN {X 0,Y 186.366,Z 91.868,A -85,B 0,C 180,E1 -22160.92,E2 -22160.92} C_VEL
LIN {X 0,Y 188.366,Z 94.176,A -85,B 0,C 180,E1 -22162.34,E2 -22162.34} C_VEL
LIN {X 0,Y 190.162,Z 95.337,A -85,B 0,C 180,E1 -22163.462,E2 -22163.462} C_VEL
LIN {X 0,Y 191.854,Z 98.388,A -85,B 0,C 180,E1 -22164.612,E2 -22164.612} C_VEL
LIN {X 0,Y 194.397,Z 100.716,A -85,B 0,C 180,E1 -22166.071,E2 -22166.071} C_VEL
LIN {X 0,Y 196.853,Z 104.288,A -85,B 0,C 180,E1 -22167.477,E2 -22167.477} C_VEL
LIN {X 0,Y 198.376,Z 105.945,A -85,B 0,C 180,E1 -22168.268,E2 -22168.268} C_VEL
LIN {X 0,Y 201.427,Z 109.919,A -85,B 0,C 180,E1 -22169.81,E2 -22169.81} C_VEL
LIN {X 0,Y 207.798,Z 118.954,A -85,B 0,C 180,E1 -22172.761,E2 -22172.761} C_VEL
LIN {X 0,Y 214.682,Z 129.542,A -85,B 0,C 180,E1 -22175.598,E2 -22175.598} C_VEL
LIN {X 0,Y 221.612,Z 141.627,A -85,B 0,C 180,E1 -22178.199,E2 -22178.199} C_VEL
LIN {X 0,Y 224.83,Z 147.708,A -85,B 0,C 180,E1 -22179.331,E2 -22179.331} C_VEL
LIN {X 0,Y 222.138,Z 189.483,A -85,B 0,C 180,E1 -22180.596,E2 -22180.596} C_VEL
LIN {X 0,Y 220.542,Z 202.628,A -85,B 0,C 180,E1 -22181.334,E2 -22181.334} C_VEL
LIN {X 0,Y 218.594,Z 214.206,A -85,B 0,C 180,E1 -22182.313,E2 -22182.313} C_VEL
LIN {X 0,Y 215.946,Z 225.401,A -85,B 0,C 180,E1 -22183.541,E2 -22183.541} C_VEL
LIN {X 0,Y 212.769,Z 236.179,A -85,B 0,C 180,E1 -22185.086,E2 -22185.086} C_VEL
LIN {X 0,Y 208.954,Z 246.957,A -85,B 0,C 180,E1 -22187.071,E2 -22187.071} C_VEL
LIN {X 0,Y 205.055,Z 256.613,A -85,B 0,C 180,E1 -22189.368,E2 -22189.368} C_VEL
LIN {X 0,Y 200.65,Z 265.819,A -85,B 0,C 180,E1 -22192.196,E2 -22192.196} C_VEL
LIN {X 0,Y 196.712,Z 273.409,A -85,B 0,C 180,E1 -22195.258,E2 -22195.258} C_VEL
LIN {X 0,Y 193.411,Z 279.035,A -85,B 0,C 180,E1 -22198.204,E2 -22198.204} C_VEL
LIN {X 0,Y 190.522,Z 283.587,A -85,B 0,C 180,E1 -22201.344,E2 -22201.344} C_VEL
LIN {X 0,Y 188.883,Z 285.964,A -85,B 0,C 180,E1 -22203.481,E2 -22203.481} C_VEL
LIN {X 0,Y 187.476,Z 287.896,A -85,B 0,C 180,E1 -22205.647,E2 -22205.647} C_VEL
LIN {X 0,Y 186.273,Z 289.397,A -85,B 0,C 180,E1 -22207.834,E2 -22207.834} C_VEL
LIN {X 0,Y 184.591,Z 291.035,A -85,B 0,C 180,E1 -22212.144,E2 -22212.144} C_VEL
LIN {X 0,Y 183.961,Z 291.3,A -85,B 0,C 180,E1 -22214.489,E2 -22214.489} C_VEL
LIN {X 0,Y 183.517,Z 291.138,A -85,B 0,C 180,E1 -22216.716,E2 -22216.716} C_VEL
LIN {X 0,Y 183.317,Z 289.548,A -85,B 0,C 180,E1 -22221.179,E2 -22221.179} C_VEL
LIN {X 0,Y 183.664,Z 287.53,A -85,B 0,C 180,E1 -22224.213,E2 -22224.213} C_VEL
LIN {X 0,Y 184.071,Z 284.079,A -85,B 0,C 180,E1 -22227.812,E2 -22227.812} C_VEL
LIN {X 0,Y 184.933,Z 279.808,A -85,B 0,C 180,E1 -22231.089,E2 -22231.089} C_VEL
LIN {X 0,Y 186.329,Z 273.367,A -85,B 0,C 180,E1 -22234.869,E2 -22234.869} C_VEL
LIN {X 0,Y 188.178,Z 266.285,A -85,B 0,C 180,E1 -22238.051,E2 -22238.051} C_VEL
LIN {X 0,Y 190.317,Z 257.487,A -85,B 0,C 180,E1 -22241.179,E2 -22241.179} C_VEL
LIN {X 0,Y 192.533,Z 248.456,A -85,B 0,C 180,E1 -22243.726,E2 -22243.726} C_VEL
LIN {X 0,Y 194.997,Z 238.438,A -85,B 0,C 180,E1 -22245.951,E2 -22245.951} C_VEL
LIN {X 0,Y 197.209,Z 227.338,A -85,B 0,C 180,E1 -22247.901,E2 -22247.901} C_VEL
LIN {X 0,Y 199.148,Z 214.948,A -85,B 0,C 180,E1 -22249.589,E2 -22249.589} C_VEL
LIN {X 0,Y 200.651,Z 202.322,A -85,B 0,C 180,E1 -22250.839,E2 -22250.839} C_VEL
LIN {X 0,Y 201.715,Z 188.927,A -85,B 0,C 180,E1 -22251.728,E2 -22251.728} C_VEL
LIN {X 0,Y 203.259,Z 154.261,A -85,B 0,C 180,E1 -22252.952,E2 -22252.952} C_VEL
LIN {X 0,Y 204.387,Z 126.949,A -85,B 0,C 180,E1 -22253.861,E2 -22253.861} C_VEL
LIN {X 0,Y 197.18,Z 111.141,A -85,B 0,C 180,E1 -22255.739,E2 -22255.739} C_VEL
LIN {X 0,Y 190.861,Z 99.369,A -85,B 0,C 180,E1 -22257.443,E2 -22257.443} C_VEL
